METHOD FB_init : BOOL
VAR_INPUT
	bInitRetains : BOOL; // if TRUE, the retain variables are initialized (warm start / cold start)
	bInCopyCode : BOOL;  // if TRUE, the instance afterwards gets moved into the copy code (online change)
END_VAR
AddInput('ipRefContour', ipRefContour);
AddInput('ipContours', ipContours);
AddParameter('fDissimilarityThreshold', fDissimilarityThreshold);
AddParameter('eComparisonMethod', eComparisonMethod);
AddParameter('fAreaFactor', fAreaFactor);
AddParameter('fAbsPositionFactor', fAbsPositionFactor);
AddInput('hrPrev', hrPrev);
AddOutput('ipMatchIndexes', ipMatchIndexes);
AddOutput('ipDissimilarities', ipDissimilarities);
AddOutput('hresult', hresult);
END_METHOD

METHOD PUBLIC  Clone : I_Node
VAR
	pNode : POINTER TO Node_F_VN_MatchContours1vsNExp;
END_VAR
pNode := __NEW(Node_F_VN_MatchContours1vsNExp);
Clone := pNode^;
END_METHOD

METHOD PROTECTED OnExecute
hresult.Value := F_VN_MatchContours1vsNExp(
	ipRefContour := ipRefContour.Value,
    ipContours := ipContours.Value,
    ipMatchIndexes := ipMatchIndexes.Value,
    ipDissimilarities := ipDissimilarities.Value,
    fDissimilarityThreshold := fDissimilarityThreshold.Value,
    eComparisonMethod := eComparisonMethod.Value,
    fAreaFactor := fAreaFactor.Value,
    fAbsPositionFactor := fAbsPositionFactor.Value,
	hrPrev:= hrPrev.Value);
END_METHOD

METHOD PUBLIC PreExecutionCheck
VAR_INPUT
	Check : I_PreExecutionChecks;
END_VAR
Check.IsTrue(ipRefContour.IsValid, 'ipRefContour must be a valid container');
Check.IsTrue((ipRefContour.IsType(TC_GLOBAL_CONST_LIST.ContainerType_Vector_TcVnPoint2_DINT) OR
              ipRefContour.IsType(TC_GLOBAL_CONST_LIST.ContainerType_Vector_TcVnPoint2_REAL)),
              'ipRefContour contains incorrect type');
              
Check.IsTrue(ipContours.IsValid, 'ipContours must be a valid container');
Check.IsTrue(ipContours.IsType(TC_GLOBAL_CONST_LIST.ContainerType_Vector_Vector_TcVnPoint2_DINT), 'ipContours contains incorrect type');

Check.IsTrue(fAreaFactor.Value >= 0, 'fAreaFactor must be greater than or equal to 0');
Check.IsTrue(fAbsPositionFactor.Value >= 0, 'fAbsPositionFactor must be greater than or equal to 0');
END_METHOD

END_FUNCTION_BLOCK

// Nodes/Contour Analysis/Node_F_VN_MatchContoursExp
{attribute 'linkalways'}
{attribute 'no_explicit_call' := 'This FB is a CLASS and must be accessed using methods or properties'}
{attribute 'enable_dynamic_creation'}
FUNCTION_BLOCK Node_F_VN_MatchContoursExp EXTENDS VisionNode
VAR
    ipContour1 : _ITcVnContainer;
    ipContour2 : _ITcVnContainer;
    eComparisonMethod : _ETcVnContoursMatchComparisonMethod(ETcVnContoursMatchComparisonMethod.TCVN_CMCM_CONTOURS_MATCH_I1);
    fDissimilarity : _LREAL(0.0);
    fAreaFactor : _LREAL(0);
    fAbsPositionFactor : _LREAL(0);
    fRelPositionFactor : _LREAL(0);
    fNumDiffFactor : _LREAL(0);
    hrPrev : _HRESULT(S_OK);
    hresult : _HRESULT(S_OK);
END_VAR

METHOD FB_init : BOOL
VAR_INPUT
    bInitRetains : BOOL;
    bInCopyCode : BOOL;
END_VAR
AddInput('ipContour1', ipContour1);
AddInput('ipContour2', ipContour2);
AddParameter('eComparisonMethod', eComparisonMethod);
AddOutput('fDissimilarity', fDissimilarity);
AddParameter('fAreaFactor', fAreaFactor);
AddParameter('fAbsPositionFactor', fAbsPositionFactor);
AddParameter('fRelPositionFactor', fRelPositionFactor);
AddParameter('fNumDiffFactor', fNumDiffFactor);
AddInput('hrPrev', hrPrev);
AddOutput('hresult', hresult);
END_METHOD

METHOD PUBLIC Clone : I_Node
VAR
    pNode : POINTER TO Node_F_VN_MatchContoursExp;
END_VAR
pNode := __NEW(Node_F_VN_MatchContoursExp);
Clone := pNode^;
END_METHOD

METHOD PROTECTED OnExecute
hresult.Value := F_VN_MatchContoursExp(
    ipContour1 := ipContour1.Value,
    ipContour2 := ipContour2.Value,
    eComparisonMethod := eComparisonMethod.Value,
    fDissimilarity := fDissimilarity.Value,
    fAreaFactor := fAreaFactor.Value,
    fAbsPositionFactor := fAbsPositionFactor.Value,
    fRelPositionFactor := fRelPositionFactor.Value,
    fNumDiffFactor := fNumDiffFactor.Value,
    hrPrev := hrPrev.Value);
END_METHOD

METHOD PUBLIC PreExecutionCheck
VAR_INPUT
    Check : I_PreExecutionChecks;
END_VAR
Check.IsTrue(ipContour1.IsValid, 'ipContour1 must contain a container');
Check.IsTrue(ipContour2.IsValid, 'ipContour2 must contain a container');
Check.IsTrue(ipContour1.IsType(TC_GLOBAL_CONST_LIST.ContainerType_Vector_TcVnPoint2_DINT) OR
             ipContour1.IsType(TC_GLOBAL_CONST_LIST.ContainerType_Vector_TcVnPoint2_REAL) OR
             ipContour1.IsType(TC_GLOBAL_CONST_LIST.ContainerType_Vector_Vector_TcVnPoint2_DINT), 'Unsupported contour container type');
Check.IsTrue(ContainersHaveMatchingTypes(ipContour1.Value, ipContour2.Value), 'Contours must have matching container types');
Check.IsTrue((eComparisonMethod.Value = ETcVnContoursMatchComparisonMethod.TCVN_CMCM_CONTOURS_MATCH_I1) OR
             (eComparisonMethod.Value = ETcVnContoursMatchComparisonMethod.TCVN_CMCM_CONTOURS_MATCH_I2) OR
             (eComparisonMethod.Value = ETcVnContoursMatchComparisonMethod.TCVN_CMCM_CONTOURS_MATCH_I3), 'Unsupported eComparisonMethod');
END_METHOD

END_FUNCTION_BLOCK

// Nodes/Contour Analysis/Node_F_VN_UprightBoundingRectangle
{attribute 'linkalways'} 
{attribute 'no_explicit_call' := 'This FB is a CLASS and must be accessed using methods or properties'}
{attribute 'enable_dynamic_creation'}
FUNCTION_BLOCK Node_F_VN_UprightBoundingRectangle EXTENDS VisionNode
VAR
    ipPointSet : _ITcVnContainer;
    stRectangle : _TcVnRectangle_UDINT;
    hrPrev : _HRESULT(S_OK);
	hresult : _HRESULT(S_OK);
END_VAR

METHOD FB_init : BOOL
VAR_INPUT
	bInitRetains : BOOL; // if TRUE, the retain variables are initialized (warm start / cold start)
	bInCopyCode : BOOL;  // if TRUE, the instance afterwards gets moved into the copy code (online change)
END_VAR
AddInput('ipPointSet', ipPointSet);
AddInput('hrPrev', hrPrev);
AddOutput('stRectangle', stRectangle);
AddOutput('hresult',hresult);
END_METHOD

METHOD PUBLIC  Clone : I_Node
VAR
	pNode : POINTER TO Node_F_VN_UprightBoundingRectangle;
END_VAR
pNode := __NEW(Node_F_VN_UprightBoundingRectangle);
Clone := pNode^;
END_METHOD

METHOD PROTECTED OnExecute
hresult.Value := F_VN_UprightBoundingRectangle(
	ipPointSet := ipPointSet.Value,
    stRectangle := stRectangle.Value,
	hrPrev:= hrPrev.Value);
END_METHOD

METHOD PUBLIC PreExecutionCheck
VAR_INPUT
	Check : I_PreExecutionChecks;
END_VAR
Check.IsTrue(ipPointSet.IsValid, 'ipPointSet must be a valid container');
Check.IsTrue((ipPointSet.IsType(TC_GLOBAL_CONST_LIST.ContainerType_Vector_TcVnPoint2_DINT) OR
              ipPointSet.IsType(TC_GLOBAL_CONST_LIST.ContainerType_Vector_TcVnPoint2_REAL)),
              'ipPointSet contains incorrect type');
END_METHOD

END_FUNCTION_BLOCK

// Nodes/Drawing/Node_F_VN_DrawArrow
{attribute 'linkalways'} 
{attribute 'no_explicit_call' := 'This FB is a CLASS and must be accessed using methods or properties'}
{attribute 'enable_dynamic_creation'}
FUNCTION_BLOCK Node_F_VN_DrawArrow EXTENDS VisionNode
VAR
    nX1 : _UDINT(0);
    nY1 : _UDINT(0);
    nX2 : _UDINT(0);
    nY2 : _UDINT(0);
    ipDestImage : _ITcVnImage;
    aColor : _TcVnVector4_LREAL;
    nThickness : _DINT(1);
    bDoubleHead : _BOOL(FALSE);
    hrPrev : _HRESULT(S_OK);
	hresult : _HRESULT(S_OK);
END_VAR

METHOD FB_init : BOOL
VAR_INPUT
	bInitRetains : BOOL; // if TRUE, the retain variables are initialized (warm start / cold start)
	bInCopyCode : BOOL;  // if TRUE, the instance afterwards gets moved into the copy code (online change)
END_VAR
AddParameter('nX1', nX1);
AddParameter('nY1', nY1);
AddParameter('nX2', nX2);
AddParameter('nY2', nY2);
AddInput('ipDestImage', ipDestImage);
AddInput('aColor', aColor);
AddParameter('nThickness', nThickness);
AddParameter('bDoubleHead', bDoubleHead);
AddInput('hrPrev', hrPrev);
AddOutput('ipDestImage', ipDestImage);
AddOutput('hresult',hresult);
END_METHOD

METHOD PUBLIC  Clone : I_Node
VAR
	pNode : POINTER TO Node_F_VN_DrawArrow;
END_VAR
pNode := __NEW(Node_F_VN_DrawArrow);
Clone := pNode^;
END_METHOD

METHOD PROTECTED OnExecute
hresult.Value := F_VN_DrawArrow(
    nX1 := nX1.Value,
    nY1 := nY1.Value,
    nX2 := nX2.Value,
    nY2 := nY2.Value,
	ipDestImage := ipDestImage.Value,
    aColor := aColor.Value,
    nThickness := nThickness.Value,
    bDoubleHead := bDoubleHead.Value,
	hrPrev:= hrPrev.Value);
END_METHOD

METHOD PUBLIC PreExecutionCheck
VAR_INPUT
	Check : I_PreExecutionChecks;
END_VAR
Check.IsTrue(ipDestImage.IsValid, 'ipDestImage must contain an image');
Check.IsTrue(nThickness.Value >= 1, 'nThickness must be greater than or equal to 1');
END_METHOD

END_FUNCTION_BLOCK

// Nodes/Drawing/Node_F_VN_DrawArrow_TcVnVector4_DINT
{attribute 'linkalways'} 
{attribute 'no_explicit_call' := 'This FB is a CLASS and must be accessed using methods or properties'}
{attribute 'enable_dynamic_creation'}
FUNCTION_BLOCK Node_F_VN_DrawArrow_TcVnVector4_DINT EXTENDS VisionNode
VAR
    aLine : _TcVnVector4_DINT;
    ipDestImage : _ITcVnImage;
    aColor : _TcVnVector4_LREAL;
    nThickness : _DINT(1);
    bDoubleHead : _BOOL(FALSE);
    hrPrev : _HRESULT(S_OK);
	hresult : _HRESULT(S_OK);
END_VAR

METHOD FB_init : BOOL
VAR_INPUT
	bInitRetains : BOOL; // if TRUE, the retain variables are initialized (warm start / cold start)
	bInCopyCode : BOOL;  // if TRUE, the instance afterwards gets moved into the copy code (online change)
END_VAR
AddInput('aLine', aLine);
AddInput('ipDestImage', ipDestImage);
AddInput('aColor', aColor);
AddParameter('nThickness', nThickness);
AddParameter('bDoubleHead', bDoubleHead);
AddInput('hrPrev', hrPrev);
AddOutput('ipDestImage', ipDestImage);
AddOutput('hresult',hresult);
END_METHOD

METHOD PUBLIC  Clone : I_Node
VAR
	pNode : POINTER TO Node_F_VN_DrawArrow_TcVnVector4_DINT;
END_VAR
pNode := __NEW(Node_F_VN_DrawArrow_TcVnVector4_DINT);
Clone := pNode^;
END_METHOD

METHOD PROTECTED OnExecute
hresult.Value := F_VN_DrawArrow_TcVnVector4_DINT(
    aLine := aLine.Value,
	ipDestImage := ipDestImage.Value,
    aColor := aColor.Value,
    nThickness := nThickness.Value,
    bDoubleHead := bDoubleHead.Value,
	hrPrev:= hrPrev.Value);
END_METHOD

METHOD PUBLIC PreExecutionCheck
VAR_INPUT
	Check : I_PreExecutionChecks;
END_VAR
Check.IsTrue(ipDestImage.IsValid, 'ipDestImage must contain an image');
Check.IsTrue(nThickness.Value >= 1, 'nThickness must be greater than or equal to 1');
END_METHOD

END_FUNCTION_BLOCK

// Nodes/Drawing/Node_F_VN_DrawArrowExp
{attribute 'linkalways'} 
{attribute 'no_explicit_call' := 'This FB is a CLASS and must be accessed using methods or properties'}
{attribute 'enable_dynamic_creation'}
FUNCTION_BLOCK Node_F_VN_DrawArrowExp EXTENDS VisionNode
VAR
    nX1 : _UDINT(0);
    nY1 : _UDINT(0);
    nX2 : _UDINT(0);
    nY2 : _UDINT(0);
    ipDestImage : _ITcVnImage;
    aColor : _TcVnVector4_LREAL;
    nThickness : _DINT(1);
    bDoubleHead : _BOOL(FALSE);
    eLineType : _ETcVnLineType(ETcVnLineType.TCVN_LT_4_CONNECTED);
    nShift : _UDINT(0);
    fTipLength : _LREAL(0.0);
    hrPrev : _HRESULT(S_OK);
	hresult : _HRESULT(S_OK);
END_VAR

METHOD FB_init : BOOL
VAR_INPUT
	bInitRetains : BOOL; // if TRUE, the retain variables are initialized (warm start / cold start)
	bInCopyCode : BOOL;  // if TRUE, the instance afterwards gets moved into the copy code (online change)
END_VAR
AddParameter('nX1', nX1);
AddParameter('nY1', nY1);
AddParameter('nX2', nX2);
AddParameter('nY2', nY2);
AddInput('ipDestImage', ipDestImage);
AddInput('aColor', aColor);
AddParameter('nThickness', nThickness);
AddParameter('bDoubleHead', bDoubleHead);
AddParameter('eLineType', eLineType);
AddParameter('nShift', nShift);
AddParameter('fTipLength', fTipLength);
AddInput('hrPrev', hrPrev);
AddOutput('ipDestImage', ipDestImage);
AddOutput('hresult', hresult);
END_METHOD

METHOD PUBLIC  Clone : I_Node
VAR
	pNode : POINTER TO Node_F_VN_DrawArrowExp;
END_VAR
pNode := __NEW(Node_F_VN_DrawArrowExp);
Clone := pNode^;
END_METHOD

METHOD PROTECTED OnExecute
hresult.Value := F_VN_DrawArrowExp(
    nX1 := nX1.Value,
    nY1 := nY1.Value,
    nX2 := nX2.Value,
    nY2 := nY2.Value,
	ipDestImage := ipDestImage.Value,
    aColor := aColor.Value,
    nThickness := nThickness.Value,
    bDoubleHead := bDoubleHead.Value,
    eLineType := eLineType.Value,
    nShift := nShift.Value,
    fTipLength := fTipLength.Value,
	hrPrev:= hrPrev.Value);
END_METHOD

METHOD PUBLIC PreExecutionCheck
VAR_INPUT
	Check : I_PreExecutionChecks;
END_VAR
Check.IsTrue(ipDestImage.IsValid, 'ipDestImage must contain an image');
Check.IsTrue(nThickness.Value >= 1, 'nThickness must be greater than or equal to 1');
END_METHOD

END_FUNCTION_BLOCK

// Nodes/Drawing/Node_F_VN_DrawArrowExp_TcVnVector4_DINT
{attribute 'linkalways'} 
{attribute 'no_explicit_call' := 'This FB is a CLASS and must be accessed using methods or properties'}
{attribute 'enable_dynamic_creation'}
FUNCTION_BLOCK Node_F_VN_DrawArrowExp_TcVnVector4_DINT EXTENDS VisionNode
VAR
    aLine : _TcVnVector4_DINT;
    ipDestImage : _ITcVnImage;
    aColor : _TcVnVector4_LREAL;
    nThickness : _DINT(1);
    bDoubleHead : _BOOL(FALSE);
    eLineType : _ETcVnLineType(ETcVnLineType.TCVN_LT_4_CONNECTED);
    nShift : _UDINT(0);
    fTipLength : _LREAL(0.0);
    hrPrev : _HRESULT(S_OK);
	hresult : _HRESULT(S_OK);
END_VAR

METHOD FB_init : BOOL
VAR_INPUT
	bInitRetains : BOOL; // if TRUE, the retain variables are initialized (warm start / cold start)
	bInCopyCode : BOOL;  // if TRUE, the instance afterwards gets moved into the copy code (online change)
END_VAR
AddInput('aLine', aLine);
AddInput('ipDestImage', ipDestImage);
AddInput('aColor', aColor);
AddParameter('nThickness', nThickness);
AddParameter('bDoubleHead', bDoubleHead);
AddParameter('eLineType', eLineType);
AddParameter('nShift', nShift);
AddParameter('fTipLength', fTipLength);
AddInput('hrPrev', hrPrev);
AddOutput('ipDestImage', ipDestImage);
AddOutput('hresult', hresult);
END_METHOD

METHOD PUBLIC  Clone : I_Node
VAR
	pNode : POINTER TO Node_F_VN_DrawArrowExp_TcVnVector4_DINT;
END_VAR
pNode := __NEW(Node_F_VN_DrawArrowExp_TcVnVector4_DINT);
Clone := pNode^;
END_METHOD

METHOD PROTECTED OnExecute
hresult.Value := F_VN_DrawArrowExp_TcVnVector4_DINT(
    aLine := aLine.Value,
	ipDestImage := ipDestImage.Value,
    aColor := aColor.Value,
    nThickness := nThickness.Value,
    bDoubleHead := bDoubleHead.Value,
    eLineType := eLineType.Value,
    nShift := nShift.Value,
    fTipLength := fTipLength.Value,
	hrPrev:= hrPrev.Value);
END_METHOD

METHOD PUBLIC PreExecutionCheck
VAR_INPUT
	Check : I_PreExecutionChecks;
END_VAR
Check.IsTrue(ipDestImage.IsValid, 'ipDestImage must contain an image');
Check.IsTrue(nThickness.Value >= 1, 'nThickness must be greater than or equal to 1');
END_METHOD

END_FUNCTION_BLOCK

// Nodes/Drawing/Node_F_VN_DrawCircle
{attribute 'linkalways'} 
{attribute 'no_explicit_call' := 'This FB is a CLASS and must be accessed using methods or properties'}
{attribute 'enable_dynamic_creation'}
FUNCTION_BLOCK Node_F_VN_DrawCircle EXTENDS VisionNode
VAR
    nCenterX : _UDINT(0);
    nCenterY : _UDINT(0);
    nRadius : _UDINT(0);
    ipDestImage : _ITcVnImage;
    aColor : _TcVnVector4_LREAL;
    nThickness : _DINT(1);
    hrPrev : _HRESULT(S_OK);
	hresult : _HRESULT(S_OK);
END_VAR

METHOD FB_init : BOOL
VAR_INPUT
	bInitRetains : BOOL; // if TRUE, the retain variables are initialized (warm start / cold start)
	bInCopyCode : BOOL;  // if TRUE, the instance afterwards gets moved into the copy code (online change)
END_VAR
AddParameter('nCenterX', nCenterX);
AddParameter('nCenterY', nCenterY);
AddParameter('nRadius', nRadius);
AddInput('ipDestImage', ipDestImage);
AddInput('aColor', aColor);
AddParameter('nThickness', nThickness);
AddInput('hrPrev', hrPrev);
AddOutput('ipDestImage', ipDestImage);
AddOutput('hresult',hresult);
END_METHOD

METHOD PUBLIC  Clone : I_Node
VAR
	pNode : POINTER TO Node_F_VN_DrawCircle;
END_VAR
pNode := __NEW(Node_F_VN_DrawCircle);
Clone := pNode^;
END_METHOD

METHOD PROTECTED OnExecute
hresult.Value := F_VN_DrawCircle(
    nCenterX := nCenterX.Value,
    nCenterY := nCenterY.Value,
    nRadius := nRadius.Value,
	ipDestImage := ipDestImage.Value,
    aColor := aColor.Value,
    nThickness := nThickness.Value,
	hrPrev:= hrPrev.Value);
END_METHOD

METHOD PUBLIC PreExecutionCheck
VAR_INPUT
	Check : I_PreExecutionChecks;
END_VAR
Check.IsTrue(ipDestImage.IsValid, 'ipDestImage must contain an image');
Check.IsTrue(nThickness.Value <> 0, 'nThickness must be non-zero');
END_METHOD

END_FUNCTION_BLOCK

// Nodes/Drawing/Node_F_VN_DrawCircleExp
{attribute 'linkalways'} 
{attribute 'no_explicit_call' := 'This FB is a CLASS and must be accessed using methods or properties'}
{attribute 'enable_dynamic_creation'}
FUNCTION_BLOCK Node_F_VN_DrawCircleExp EXTENDS VisionNode
VAR
    nCenterX : _UDINT(0);
    nCenterY : _UDINT(0);
    nRadius : _UDINT(0);
    ipDestImage : _ITcVnImage;
    aColor : _TcVnVector4_LREAL;
    nThickness : _DINT(1);
    eLineType : _ETcVnLineType(ETcVnLineType.TCVN_LT_4_CONNECTED);
    hrPrev : _HRESULT(S_OK);
	hresult : _HRESULT(S_OK);
END_VAR

METHOD FB_init : BOOL
VAR_INPUT
	bInitRetains : BOOL; // if TRUE, the retain variables are initialized (warm start / cold start)
	bInCopyCode : BOOL;  // if TRUE, the instance afterwards gets moved into the copy code (online change)
END_VAR
AddParameter('nCenterX', nCenterX);
AddParameter('nCenterY', nCenterY);
AddParameter('nRadius', nRadius);
AddInput('ipDestImage', ipDestImage);
AddInput('aColor', aColor);
AddParameter('nThickness', nThickness);
AddParameter('eLineType', eLineType);
AddInput('hrPrev', hrPrev);
AddOutput('ipDestImage', ipDestImage);
AddOutput('hresult',hresult);
END_METHOD

METHOD PUBLIC  Clone : I_Node
VAR
	pNode : POINTER TO Node_F_VN_DrawCircleExp;
END_VAR
pNode := __NEW(Node_F_VN_DrawCircleExp);
Clone := pNode^;
END_METHOD

METHOD PROTECTED OnExecute
hresult.Value := F_VN_DrawCircleExp(
    nCenterX := nCenterX.Value,
    nCenterY := nCenterY.Value,
    nRadius := nRadius.Value,
	ipDestImage := ipDestImage.Value,
    aColor := aColor.Value,
    nThickness := nThickness.Value,
    eLineType := eLineType.Value,
	hrPrev:= hrPrev.Value);
END_METHOD

METHOD PUBLIC PreExecutionCheck
VAR_INPUT
	Check : I_PreExecutionChecks;
END_VAR
Check.IsTrue(ipDestImage.IsValid, 'ipDestImage must contain an image');
Check.IsTrue(nThickness.Value <> 0, 'nThickness must be non-zero');
END_METHOD

END_FUNCTION_BLOCK

// Nodes/Drawing/Node_F_VN_DrawCircles
{attribute 'linkalways'} 
{attribute 'no_explicit_call' := 'This FB is a CLASS and must be accessed using methods or properties'}
{attribute 'enable_dynamic_creation'}
FUNCTION_BLOCK Node_F_VN_DrawCircles EXTENDS VisionNode
VAR
    ipCircles : _ITcVnContainer;
    nCircleIndex : _DINT(0);
    ipDestImage : _ITcVnImage;
    aColor : _TcVnVector4_LREAL;
    nThickness : _DINT(1);
    hrPrev : _HRESULT(S_OK);
	hresult : _HRESULT(S_OK);
END_VAR

METHOD FB_init : BOOL
VAR_INPUT
	bInitRetains : BOOL; // if TRUE, the retain variables are initialized (warm start / cold start)
	bInCopyCode : BOOL;  // if TRUE, the instance afterwards gets moved into the copy code (online change)
END_VAR
AddInput('ipCircles', ipCircles);
AddParameter('nCircleIndex', nCircleIndex);
AddInput('ipDestImage', ipDestImage);
AddInput('aColor', aColor);
AddParameter('nThickness', nThickness);
AddInput('hrPrev', hrPrev);
AddOutput('ipDestImage', ipDestImage);
AddOutput('hresult',hresult);
END_METHOD

METHOD PUBLIC  Clone : I_Node
VAR
	pNode : POINTER TO Node_F_VN_DrawCircles
;
END_VAR
pNode := __NEW(Node_F_VN_DrawCircles);
Clone := pNode^;
END_METHOD

METHOD PROTECTED OnExecute
hresult.Value := F_VN_DrawCircles(
    ipCircles := ipCircles.Value,
    nCircleIndex := nCircleIndex.Value,
	ipDestImage := ipDestImage.Value,
    aColor := aColor.Value,
    nThickness := nThickness.Value,
	hrPrev:= hrPrev.Value);
END_METHOD

METHOD PUBLIC PreExecutionCheck
VAR_INPUT
	Check : I_PreExecutionChecks;
END_VAR
VAR
    containerElements : ULINT;
    maxIndexNumber : ULINT;
END_VAR
Check.IsTrue(ipCircles.IsValid, 'ipCircles must be a valid container');
Check.IsTrue(ipCircles.IsType(TC_GLOBAL_CONST_LIST.ContainerType_Vector_TcVnVector3_REAL), 'ipCircles contains incorrect type');

Check.IsTrue(ipCircles.TryGetElementNum(containerElements) AND (containerElements > 0), 'ipCircles is empty');

IF Check.Failed THEN
    RETURN;
END_IF

maxIndexNumber := containerElements - 1;

IF (nCircleIndex.Value > -1) THEN
    Check.IsTrue((DINT_TO_ULINT(nCircleIndex.Value) <= maxIndexNumber), 'nCircleIndex out of range.');
END_IF

Check.IsTrue(ipDestImage.IsValid, 'ipDestImage must contain an image');
Check.IsTrue(nThickness.Value <> 0, 'nThickness must be non-zero');
END_METHOD

END_FUNCTION_BLOCK

// Nodes/Drawing/Node_F_VN_DrawCirclesExp
{attribute 'linkalways'} 
{attribute 'no_explicit_call' := 'This FB is a CLASS and must be accessed using methods or properties'}
{attribute 'enable_dynamic_creation'}
FUNCTION_BLOCK Node_F_VN_DrawCirclesExp EXTENDS VisionNode
VAR
    ipCircles : _ITcVnContainer;
    nCircleIndex : _DINT(0);
    ipDestImage : _ITcVnImage;
    aColor : _TcVnVector4_LREAL;
    nThickness : _DINT(1);
    eLineType : _ETcVnLineType(ETcVnLineType.TCVN_LT_4_CONNECTED);
    hrPrev : _HRESULT(S_OK);
	hresult : _HRESULT(S_OK);
END_VAR

METHOD FB_init : BOOL
VAR_INPUT
	bInitRetains : BOOL; // if TRUE, the retain variables are initialized (warm start / cold start)
	bInCopyCode : BOOL;  // if TRUE, the instance afterwards gets moved into the copy code (online change)
END_VAR
AddInput('ipCircles', ipCircles);
AddParameter('nCircleIndex', nCircleIndex);
AddInput('ipDestImage', ipDestImage);
AddInput('aColor', aColor);
AddParameter('nThickness', nThickness);
AddParameter('eLineType', eLineType);
AddInput('hrPrev', hrPrev);
AddOutput('ipDestImage', ipDestImage);
AddOutput('hresult',hresult);
END_METHOD

METHOD PUBLIC  Clone : I_Node
VAR
	pNode : POINTER TO Node_F_VN_DrawCirclesExp
;
END_VAR
pNode := __NEW(Node_F_VN_DrawCirclesExp);
Clone := pNode^;
END_METHOD

METHOD PROTECTED OnExecute
hresult.Value := F_VN_DrawCirclesExp(
    ipCircles := ipCircles.Value,
    nCircleIndex := nCircleIndex.Value,
	ipDestImage := ipDestImage.Value,
    aColor := aColor.Value,
    nThickness := nThickness.Value,
    eLineType := eLineType.Value,
	hrPrev:= hrPrev.Value);
END_METHOD

METHOD PUBLIC PreExecutionCheck
VAR_INPUT
	Check : I_PreExecutionChecks;
END_VAR
VAR
    containerElements : ULINT;
    maxIndexNumber : ULINT;
END_VAR
Check.IsTrue(ipCircles.IsValid, 'ipCircles must be a valid container');
Check.IsTrue(ipCircles.IsType(TC_GLOBAL_CONST_LIST.ContainerType_Vector_TcVnVector3_REAL), 'ipCircles contains incorrect type');

Check.IsTrue(ipCircles.TryGetElementNum(containerElements) AND (containerElements > 0), 'ipCircles is empty');

IF Check.Failed THEN
    RETURN;
END_IF

maxIndexNumber := containerElements - 1;

IF (nCircleIndex.Value > -1) THEN
    Check.IsTrue((DINT_TO_ULINT(nCircleIndex.Value) <= maxIndexNumber), 'nCircleIndex out of range.');
END_IF

Check.IsTrue(ipDestImage.IsValid, 'ipDestImage must contain an image');
Check.IsTrue(nThickness.Value <> 0, 'nThickness must be non-zero');
END_METHOD

END_FUNCTION_BLOCK

// Nodes/Drawing/Node_F_VN_DrawCircularArc
{attribute 'linkalways'} 
{attribute 'no_explicit_call' := 'This FB is a CLASS and must be accessed using methods or properties'}
{attribute 'enable_dynamic_creation'}
FUNCTION_BLOCK Node_F_VN_DrawCircularArc EXTENDS VisionNode
VAR
    stCircularArc : _TcVnCircularArc;
    ipDestImage : _ITcVnImage;
    aColor : _TcVnVector4_LREAL;
    nThickness : _DINT(1);
    hrPrev : _HRESULT(S_OK);
	hresult : _HRESULT(S_OK);
END_VAR

METHOD FB_init : BOOL
VAR_INPUT
	bInitRetains : BOOL; // if TRUE, the retain variables are initialized (warm start / cold start)
	bInCopyCode : BOOL;  // if TRUE, the instance afterwards gets moved into the copy code (online change)
END_VAR
AddInput('stCircularArc', stCircularArc);
AddInput('ipDestImage', ipDestImage);
AddInput('aColor', aColor);
AddParameter('nThickness', nThickness);
AddInput('hrPrev', hrPrev);
AddOutput('ipDestImage', ipDestImage);
AddOutput('hresult',hresult);
END_METHOD

METHOD PUBLIC  Clone : I_Node
VAR
	pNode : POINTER TO Node_F_VN_DrawCircularArc;
END_VAR
pNode := __NEW(Node_F_VN_DrawCircularArc);
Clone := pNode^;
END_METHOD

METHOD PROTECTED OnExecute
hresult.Value := F_VN_DrawCircularArc(
    stCircularArc := stCircularArc.Value,
	ipDestImage := ipDestImage.Value,
    aColor := aColor.Value,
    nThickness := nThickness.Value,
	hrPrev:= hrPrev.Value);
END_METHOD

METHOD PUBLIC PreExecutionCheck
VAR_INPUT
	Check : I_PreExecutionChecks;
END_VAR
Check.IsTrue(ipDestImage.IsValid, 'ipDestImage must contain an image');
Check.IsTrue(nThickness.Value <> 0, 'nThickness must be non-zero');
END_METHOD

END_FUNCTION_BLOCK

// Nodes/Drawing/Node_F_VN_DrawCircularArcExp
{attribute 'linkalways'} 
{attribute 'no_explicit_call' := 'This FB is a CLASS and must be accessed using methods or properties'}
{attribute 'enable_dynamic_creation'}
FUNCTION_BLOCK Node_F_VN_DrawCircularArcExp EXTENDS VisionNode
VAR
    stCircularArc : _TcVnCircularArc;
    ipDestImage : _ITcVnImage;
    aColor : _TcVnVector4_LREAL;
    nThickness : _DINT(1);
    eLineType : _ETcVnLineType(ETcVnLineType.TCVN_LT_4_CONNECTED);
    hrPrev : _HRESULT(S_OK);
	hresult : _HRESULT(S_OK);
END_VAR

METHOD FB_init : BOOL
VAR_INPUT
	bInitRetains : BOOL; // if TRUE, the retain variables are initialized (warm start / cold start)
	bInCopyCode : BOOL;  // if TRUE, the instance afterwards gets moved into the copy code (online change)
END_VAR
AddInput('stCircularArc', stCircularArc);
AddInput('ipDestImage', ipDestImage);
AddInput('aColor', aColor);
AddParameter('nThickness', nThickness);
AddParameter('eLineType', eLineType);
AddInput('hrPrev', hrPrev);
AddOutput('ipDestImage', ipDestImage);
AddOutput('hresult',hresult);
END_METHOD

METHOD PUBLIC  Clone : I_Node
VAR
	pNode : POINTER TO Node_F_VN_DrawCircularArcExp;
END_VAR
pNode := __NEW(Node_F_VN_DrawCircularArcExp);
Clone := pNode^;
END_METHOD

METHOD PROTECTED OnExecute
hresult.Value := F_VN_DrawCircularArcExp(
    stCircularArc := stCircularArc.Value,
	ipDestImage := ipDestImage.Value,
    aColor := aColor.Value,
    nThickness := nThickness.Value,
    eLineType := eLineType.Value,
	hrPrev:= hrPrev.Value);
END_METHOD

METHOD PUBLIC PreExecutionCheck
VAR_INPUT
	Check : I_PreExecutionChecks;
END_VAR
Check.IsTrue(ipDestImage.IsValid, 'ipDestImage must contain an image');
Check.IsTrue(nThickness.Value <> 0, 'nThickness must be non-zero');
END_METHOD

END_FUNCTION_BLOCK

// Nodes/Drawing/Node_F_VN_DrawComponents
{attribute 'linkalways'} 
{attribute 'no_explicit_call' := 'This FB is a CLASS and must be accessed using methods or properties'}
{attribute 'enable_dynamic_creation'}
FUNCTION_BLOCK Node_F_VN_DrawComponents EXTENDS VisionNode
VAR
    ipLabelImage : _ITcVnImage;
    nLabelID : _DINT(0);
    ipDestImage : _ITcVnImage;
    bShowLabelID : _BOOL(FALSE);
    hrPrev : _HRESULT(S_OK);
	hresult : _HRESULT(S_OK);
END_VAR

METHOD FB_init : BOOL
VAR_INPUT
	bInitRetains : BOOL; // if TRUE, the retain variables are initialized (warm start / cold start)
	bInCopyCode : BOOL;  // if TRUE, the instance afterwards gets moved into the copy code (online change)
END_VAR
AddInput('ipLabelImage', ipLabelImage);
AddParameter('nLabelID', nLabelID);
AddParameter('bShowLabelID', bShowLabelID);
AddInput('hrPrev', hrPrev);
AddOutput('ipDestImage', ipDestImage);
AddOutput('hresult',hresult);
END_METHOD

METHOD PUBLIC  Clone : I_Node
VAR
	pNode : POINTER TO Node_F_VN_DrawComponents;
END_VAR
pNode := __NEW(Node_F_VN_DrawComponents);
Clone := pNode^;
END_METHOD

METHOD PROTECTED OnExecute
hresult.Value := F_VN_DrawComponents(
	ipLabelImage := ipLabelImage.Value,
    nLabelID := nLabelID.Value,
    ipDestImage := ipDestImage.Value,
    bShowLabelID := bShowLabelID.Value,
	hrPrev:= hrPrev.Value);
END_METHOD

METHOD PUBLIC PreExecutionCheck
VAR_INPUT
	Check : I_PreExecutionChecks;
END_VAR
Check.IsTrue(ipLabelImage.IsValid, 'ipLabelImage must contain an image');
Check.IsTrue(ipLabelImage.HasChannelCount(1), 'ipLabelImage must have 1 channel');
Check.IsTrue((ipLabelImage.IsPixelDepth(16)  OR
              ipLabelImage.IsPixelDepth(32)), 'ipLabelImage must have 16 or 32 bit pixel depth');
END_METHOD

END_FUNCTION_BLOCK

// Nodes/Drawing/Node_F_VN_DrawComponentsExp
{attribute 'linkalways'} 
{attribute 'no_explicit_call' := 'This FB is a CLASS and must be accessed using methods or properties'}
{attribute 'enable_dynamic_creation'}
FUNCTION_BLOCK Node_F_VN_DrawComponentsExp EXTENDS VisionNode
VAR
    ipLabelImage : _ITcVnImage;
    nLabelID : _DINT(0);
    ipDestImage : _ITcVnImage;
    bShowLabelID : _BOOL(FALSE);
    aColor : _TcVnVector4_LREAL;
    nThickness : _DINT(1);
    fFontScale : _LREAL(1.0);
    hrPrev : _HRESULT(S_OK);
	hresult : _HRESULT(S_OK);
END_VAR

METHOD FB_init : BOOL
VAR_INPUT
	bInitRetains : BOOL; // if TRUE, the retain variables are initialized (warm start / cold start)
	bInCopyCode : BOOL;  // if TRUE, the instance afterwards gets moved into the copy code (online change)
END_VAR
AddInput('ipLabelImage', ipLabelImage);
AddParameter('nLabelID', nLabelID);
AddInput('bShowLabelID', bShowLabelID);
AddInput('aColor', aColor);
AddParameter('nThickness', nThickness);
AddParameter('fFontScale', fFontScale);
AddInput('hrPrev', hrPrev);
AddOutput('ipDestImage', ipDestImage);
AddOutput('hresult',hresult);
END_METHOD

METHOD PUBLIC  Clone : I_Node
VAR
	pNode : POINTER TO Node_F_VN_DrawComponentsExp;
END_VAR
pNode := __NEW(Node_F_VN_DrawComponentsExp);
Clone := pNode^;
END_METHOD

METHOD PROTECTED OnExecute
hresult.Value := F_VN_DrawComponentsExp(
	ipLabelImage := ipLabelImage.Value,
    nLabelID := nLabelID.Value,
    ipDestImage := ipDestImage.Value,
    bShowLabelID := bShowLabelID.Value,
    aColor := aColor.Value,
    nThickness := nThickness.Value,
    fFontScale := fFontScale.Value,
	hrPrev:= hrPrev.Value);
END_METHOD

METHOD PUBLIC PreExecutionCheck
VAR_INPUT
	Check : I_PreExecutionChecks;
END_VAR
Check.IsTrue(ipLabelImage.IsValid, 'ipLabelImage must contain an image');
Check.IsTrue(ipLabelImage.HasChannelCount(1), 'ipLabelImage must have 1 channel');
Check.IsTrue((ipLabelImage.IsPixelDepth(16)  OR
              ipLabelImage.IsPixelDepth(32)), 'ipLabelImage must have 16 or 32 bit pixel depth');
Check.IsTrue(nThickness.Value >= 1, 'nThickness must be greater than or equal to 1');
END_METHOD

END_FUNCTION_BLOCK

// Nodes/Drawing/Node_F_VN_DrawContours
{attribute 'linkalways'} 
{attribute 'no_explicit_call' := 'This FB is a CLASS and must be accessed using methods or properties'}
{attribute 'enable_dynamic_creation'}
FUNCTION_BLOCK Node_F_VN_DrawContours EXTENDS VisionNode
VAR
    ipContours : _ITcVnContainer;
    nContourIndex : _DINT(0);
    ipDestImage : _ITcVnImage;
    aColor : _TcVnVector4_LREAL;
    nThickness : _DINT(1);
    hrPrev : _HRESULT(S_OK);
	hresult : _HRESULT(S_OK);
END_VAR

METHOD FB_init : BOOL
VAR_INPUT
	bInitRetains : BOOL; // if TRUE, the retain variables are initialized (warm start / cold start)
	bInCopyCode : BOOL;  // if TRUE, the instance afterwards gets moved into the copy code (online change)
END_VAR
AddInput('ipContours', ipContours);
AddParameter('nContourIndex', nContourIndex);
AddInput('ipDestImage', ipDestImage);
AddInput('aColor', aColor);
AddParameter('nThickness', nThickness);
AddInput('hrPrev', hrPrev);
AddOutput('ipDestImage', ipDestImage);
AddOutput('hresult',hresult);
END_METHOD

METHOD PUBLIC  Clone : I_Node
VAR
	pNode : POINTER TO Node_F_VN_DrawContours
;
END_VAR
pNode := __NEW(Node_F_VN_DrawContours);
Clone := pNode^;
END_METHOD

METHOD PROTECTED OnExecute
hresult.Value := F_VN_DrawContours(
    ipContours := ipContours.Value,
    nContourIndex := nContourIndex.Value,
	ipDestImage := ipDestImage.Value,
    aColor := aColor.Value,
    nThickness := nThickness.Value,
	hrPrev:= hrPrev.Value);
END_METHOD

METHOD PUBLIC PreExecutionCheck
VAR_INPUT
	Check : I_PreExecutionChecks;
END_VAR
VAR
    containerElements : ULINT;
    maxIndexNumber : ULINT;
END_VAR
Check.IsTrue(ipContours.IsValid, 'ipContours must be a valid container');
Check.IsTrue((ipContours.IsType(TC_GLOBAL_CONST_LIST.ContainerType_Vector_TcVnPoint2_DINT) OR
              ipContours.IsType(TC_GLOBAL_CONST_LIST.ContainerType_Vector_Vector_TcVnPoint2_DINT)),
              'ipContours contains incorrect type');

Check.IsTrue(ipDestImage.IsValid, 'ipDestImage must contain an image');
Check.IsTrue(nThickness.Value <> 0, 'nThickness must be non-zero');
END_METHOD

END_FUNCTION_BLOCK

// Nodes/Drawing/Node_F_VN_DrawContoursExp
{attribute 'linkalways'} 
{attribute 'no_explicit_call' := 'This FB is a CLASS and must be accessed using methods or properties'}
{attribute 'enable_dynamic_creation'}
FUNCTION_BLOCK Node_F_VN_DrawContoursExp EXTENDS VisionNode
VAR
    ipContours : _ITcVnContainer;
    nContourIndex : _DINT(0);
    ipDestImage : _ITcVnImage;
    aColor : _TcVnVector4_LREAL;
    nThickness : _DINT(1);
    eLineType : _ETcVnLineType(ETcVnLineType.TCVN_LT_4_CONNECTED);
    ipHierarchy : _ITcVnContainer;
    nMaxLevel : _DINT(0);
    aOffset : _TcVnPoint;
    hrPrev : _HRESULT(S_OK);
	hresult : _HRESULT(S_OK);
END_VAR

METHOD FB_init : BOOL
VAR_INPUT
	bInitRetains : BOOL; // if TRUE, the retain variables are initialized (warm start / cold start)
	bInCopyCode : BOOL;  // if TRUE, the instance afterwards gets moved into the copy code (online change)
END_VAR
AddInput('ipContours', ipContours);
AddParameter('nContourIndex', nContourIndex);
AddInput('ipDestImage', ipDestImage);
AddInput('aColor', aColor);
AddParameter('nThickness', nThickness);
AddParameter('eLineType', eLineType);
AddInput('ipHierarchy', ipHierarchy);
AddParameter('nMaxLevel', nMaxLevel);
AddInput('aOffset', aOffset);
AddInput('hrPrev', hrPrev);
AddOutput('ipDestImage', ipDestImage);
AddOutput('hresult',hresult);
END_METHOD

METHOD PUBLIC  Clone : I_Node
VAR
	pNode : POINTER TO Node_F_VN_DrawContoursExp
;
END_VAR
pNode := __NEW(Node_F_VN_DrawContoursExp);
Clone := pNode^;
END_METHOD

METHOD PROTECTED OnExecute
hresult.Value := F_VN_DrawContoursExp(
    ipContours := ipContours.Value,
    nContourIndex := nContourIndex.Value,
	ipDestImage := ipDestImage.Value,
    aColor := aColor.Value,
    nThickness := nThickness.Value,
    eLineType := eLineType.Value,
    ipHierarchy := ipHierarchy.Value,
    nMaxLevel := nMaxLevel.Value,
    aOffset := aOffset.Value,
	hrPrev:= hrPrev.Value);
END_METHOD

METHOD PUBLIC PreExecutionCheck
VAR_INPUT
	Check : I_PreExecutionChecks;
END_VAR
VAR
    containerElements : ULINT;
    maxIndexNumber : ULINT;
END_VAR
Check.IsTrue(ipContours.IsValid, 'ipContours must be a valid container');
Check.IsTrue((ipContours.IsType(TC_GLOBAL_CONST_LIST.ContainerType_Vector_TcVnPoint2_DINT) OR
              ipContours.IsType(TC_GLOBAL_CONST_LIST.ContainerType_Vector_Vector_TcVnPoint2_DINT)),
              'ipContours contains incorrect type');

Check.IsTrue(ipDestImage.IsValid, 'ipDestImage must contain an image');
Check.IsTrue(nThickness.Value <> 0, 'nThickness must be non-zero');
END_METHOD

END_FUNCTION_BLOCK

// Nodes/Drawing/Node_F_VN_DrawEllipse
{attribute 'linkalways'} 
{attribute 'no_explicit_call' := 'This FB is a CLASS and must be accessed using methods or properties'}
{attribute 'enable_dynamic_creation'}
FUNCTION_BLOCK Node_F_VN_DrawEllipse EXTENDS VisionNode
VAR
    stEllipse : _TcVnRotatedRectangle;
    ipDestImage : _ITcVnImage;
    aColor : _TcVnVector4_LREAL;
    nThickness : _DINT(1);
    hrPrev : _HRESULT(S_OK);
	hresult : _HRESULT(S_OK);
END_VAR

METHOD FB_init : BOOL
VAR_INPUT
	bInitRetains : BOOL; // if TRUE, the retain variables are initialized (warm start / cold start)
	bInCopyCode : BOOL;  // if TRUE, the instance afterwards gets moved into the copy code (online change)
END_VAR
AddInput('stEllipse', stEllipse);
AddInput('ipDestImage', ipDestImage);
AddInput('aColor', aColor);
AddInput('hrPrev', hrPrev);
AddOutput('ipDestImage', ipDestImage);
AddOutput('hresult',hresult);
AddParameter('nThickness', nThickness);
END_METHOD

METHOD PUBLIC  Clone : I_Node
VAR
	pNode : POINTER TO Node_F_VN_DrawEllipse;
END_VAR
pNode := __NEW(Node_F_VN_DrawEllipse);
Clone := pNode^;
END_METHOD

METHOD PROTECTED OnExecute
hresult.Value := F_VN_DrawEllipse(
    stEllipse := stEllipse.Value,
	ipDestImage := ipDestImage.Value,
    aColor := aColor.Value,
    nThickness := nThickness.Value,
	hrPrev:= hrPrev.Value);
END_METHOD

METHOD PUBLIC PreExecutionCheck
VAR_INPUT
	Check : I_PreExecutionChecks;
END_VAR
Check.IsTrue(ipDestImage.IsValid, 'ipDestImage must contain an image');
Check.IsTrue(nThickness.Value <> 0, 'nThickness must be non-zero');
END_METHOD

END_FUNCTION_BLOCK

// Nodes/Drawing/Node_F_VN_DrawEllipseExp
{attribute 'linkalways'} 
{attribute 'no_explicit_call' := 'This FB is a CLASS and must be accessed using methods or properties'}
{attribute 'enable_dynamic_creation'}
FUNCTION_BLOCK Node_F_VN_DrawEllipseExp EXTENDS VisionNode
VAR
    stEllipse : _TcVnRotatedRectangle;
    ipDestImage : _ITcVnImage;
    aColor : _TcVnVector4_LREAL;
    nThickness : _DINT(1);
    eLineType : _ETcVnLineType(ETcVnLineType.TCVN_LT_4_CONNECTED);
    hrPrev : _HRESULT(S_OK);
	hresult : _HRESULT(S_OK);
END_VAR

METHOD FB_init : BOOL
VAR_INPUT
	bInitRetains : BOOL; // if TRUE, the retain variables are initialized (warm start / cold start)
	bInCopyCode : BOOL;  // if TRUE, the instance afterwards gets moved into the copy code (online change)
END_VAR
AddInput('stEllipse', stEllipse);
AddInput('ipDestImage', ipDestImage);
AddInput('aColor', aColor);
AddParameter('nThickness', nThickness);
AddParameter('eLineType', eLineType);
AddInput('hrPrev', hrPrev);
AddOutput('ipDestImage', ipDestImage);
AddOutput('hresult',hresult);
END_METHOD

METHOD PUBLIC  Clone : I_Node
VAR
	pNode : POINTER TO Node_F_VN_DrawEllipseExp;
END_VAR
pNode := __NEW(Node_F_VN_DrawEllipseExp);
Clone := pNode^;
END_METHOD

METHOD PROTECTED OnExecute
hresult.Value := F_VN_DrawEllipseExp(
    stEllipse := stEllipse.Value,
	ipDestImage := ipDestImage.Value,
    aColor := aColor.Value,
    nThickness := nThickness.Value,
    eLineType := eLineType.Value,
	hrPrev:= hrPrev.Value);
END_METHOD

METHOD PUBLIC PreExecutionCheck
VAR_INPUT
	Check : I_PreExecutionChecks;
END_VAR
Check.IsTrue(ipDestImage.IsValid, 'ipDestImage must contain an image');
Check.IsTrue(nThickness.Value <> 0, 'nThickness must be non-zero');
END_METHOD

END_FUNCTION_BLOCK

// Nodes/Drawing/Node_F_VN_DrawKeypoints
{attribute 'linkalways'} 
{attribute 'no_explicit_call' := 'This FB is a CLASS and must be accessed using methods or properties'}
{attribute 'enable_dynamic_creation'}
FUNCTION_BLOCK Node_F_VN_DrawKeypoints EXTENDS VisionNode
VAR
    ipSrcImage : _ITcVnImage;
    ipKeyPoints : _ITcVnContainer;
    ipDestImage : _ITcVnImage;
    hrPrev : _HRESULT(S_OK);
	hresult : _HRESULT(S_OK);
END_VAR

METHOD FB_init : BOOL
VAR_INPUT
	bInitRetains : BOOL; // if TRUE, the retain variables are initialized (warm start / cold start)
	bInCopyCode : BOOL;  // if TRUE, the instance afterwards gets moved into the copy code (online change)
END_VAR
AddInput('ipSrcImage', ipSrcImage);
AddInput('ipKeyPoints', ipKeyPoints);
AddInput('hrPrev', hrPrev);
AddOutput('ipDestImage', ipDestImage);
AddOutput('hresult',hresult);
END_METHOD

METHOD PUBLIC  Clone : I_Node
VAR
	pNode : POINTER TO Node_F_VN_DrawKeypoints
;
END_VAR
pNode := __NEW(Node_F_VN_DrawKeypoints);
Clone := pNode^;
END_METHOD

METHOD PROTECTED OnExecute
hresult.Value := F_VN_DrawKeypoints(
    ipSrcImage := ipSrcImage.Value,
    ipKeyPoints := ipKeyPoints.Value,
	ipDestImage := ipDestImage.Value,
	hrPrev:= hrPrev.Value);
END_METHOD

METHOD PUBLIC PreExecutionCheck
VAR_INPUT
	Check : I_PreExecutionChecks;
END_VAR
Check.IsTrue(ipSrcImage.IsValid, 'ipSrcImage must contain an image');
Check.IsTrue(ipKeyPoints.IsType(TC_GLOBAL_CONST_LIST.ContainerType_Vector_TcVnKeyPoint), 'ipKeyPoints contains incorrect type');
END_METHOD

END_FUNCTION_BLOCK

// Nodes/Drawing/Node_F_VN_DrawKeypointsExp
{attribute 'linkalways'} 
{attribute 'no_explicit_call' := 'This FB is a CLASS and must be accessed using methods or properties'}
{attribute 'enable_dynamic_creation'}
FUNCTION_BLOCK Node_F_VN_DrawKeypointsExp EXTENDS VisionNode
VAR
    ipSrcImage : _ITcVnImage;
    ipKeyPoints : _ITcVnContainer;
    ipDestImage : _ITcVnImage;
    aColor : _TcVnVector4_LREAL;
    eFlags : _ETcVnDrawMatchesFlags(ETcVnDrawMatchesFlags.TCVN_DMF_DEFAULT);
    hrPrev : _HRESULT(S_OK);
	hresult : _HRESULT(S_OK);
END_VAR

METHOD FB_init : BOOL
VAR_INPUT
	bInitRetains : BOOL; // if TRUE, the retain variables are initialized (warm start / cold start)
	bInCopyCode : BOOL;  // if TRUE, the instance afterwards gets moved into the copy code (online change)
END_VAR
AddInput('ipSrcImage', ipSrcImage);
AddInput('ipKeyPoints', ipKeyPoints);
AddInput('aColor', aColor);
AddParameter('eFlags', eFlags);
AddInput('hrPrev', hrPrev);
AddOutput('ipDestImage', ipDestImage);
AddOutput('hresult',hresult);
END_METHOD

METHOD PUBLIC  Clone : I_Node
VAR
	pNode : POINTER TO Node_F_VN_DrawKeypointsExp
;
END_VAR
pNode := __NEW(Node_F_VN_DrawKeypointsExp);
Clone := pNode^;
END_METHOD

METHOD PROTECTED OnExecute
hresult.Value := F_VN_DrawKeypointsExp(
    ipSrcImage := ipSrcImage.Value,
    ipKeyPoints := ipKeyPoints.Value,
	ipDestImage := ipDestImage.Value,
    aColor := aColor.Value,
    eFlags := eFlags.Value,
	hrPrev:= hrPrev.Value);
END_METHOD

METHOD PUBLIC PreExecutionCheck
VAR_INPUT
	Check : I_PreExecutionChecks;
END_VAR
Check.IsTrue(ipSrcImage.IsValid, 'ipSrcImage must contain an image');
Check.IsTrue(ipSrcImage.IsPixelDepth(8), 'ipSrcImage must have 8 bit pixel depth');
Check.IsTrue(ipKeyPoints.IsType(TC_GLOBAL_CONST_LIST.ContainerType_Vector_TcVnKeyPoint), 'ipKeyPoints contains incorrect type');
END_METHOD

END_FUNCTION_BLOCK

// Nodes/Drawing/Node_F_VN_DrawLine
{attribute 'linkalways'} 
{attribute 'no_explicit_call' := 'This FB is a CLASS and must be accessed using methods or properties'}
{attribute 'enable_dynamic_creation'}
FUNCTION_BLOCK Node_F_VN_DrawLine EXTENDS VisionNode
VAR
    nX1 : _UDINT(0);
    nY1 : _UDINT(0);
    nX2 : _UDINT(0);
    nY2 : _UDINT(0);
    ipDestImage : _ITcVnImage;
    aColor : _TcVnVector4_LREAL;
    nThickness : _DINT(1);
    hrPrev : _HRESULT(S_OK);
	hresult : _HRESULT(S_OK);
END_VAR

METHOD FB_init : BOOL
VAR_INPUT
	bInitRetains : BOOL; // if TRUE, the retain variables are initialized (warm start / cold start)
	bInCopyCode : BOOL;  // if TRUE, the instance afterwards gets moved into the copy code (online change)
END_VAR
AddParameter('nX1', nX1);
AddParameter('nY1', nY1);
AddParameter('nX2', nX2);
AddParameter('nY2', nY2);
AddInput('ipDestImage', ipDestImage);
AddInput('aColor', aColor);
AddParameter('nThickness', nThickness);
AddInput('hrPrev', hrPrev);
AddOutput('ipDestImage', ipDestImage);
AddOutput('hresult',hresult);
END_METHOD

METHOD PUBLIC  Clone : I_Node
VAR
	pNode : POINTER TO Node_F_VN_DrawLine;
END_VAR
pNode := __NEW(Node_F_VN_DrawLine);
Clone := pNode^;
END_METHOD

METHOD PROTECTED OnExecute
hresult.Value := F_VN_DrawLine(
    nX1 := nX1.Value,
    nY1 := nY1.Value,
    nX2 := nX2.Value,
	nY2 := nY2.Value,
	ipDestImage := ipDestImage.Value,
    aColor := aColor.Value,
    nThickness := nThickness.Value,
	hrPrev:= hrPrev.Value);
END_METHOD

METHOD PUBLIC PreExecutionCheck
VAR_INPUT
	Check : I_PreExecutionChecks;
END_VAR
Check.IsTrue(ipDestImage.IsValid, 'ipDestImage must contain an image');
Check.IsTrue(nThickness.Value >= 1, 'nThickness must be greater than or equal to 1');
END_METHOD

END_FUNCTION_BLOCK

// Nodes/Drawing/Node_F_VN_DrawLine_TcVnVector4_DINT
{attribute 'linkalways'} 
{attribute 'no_explicit_call' := 'This FB is a CLASS and must be accessed using methods or properties'}
{attribute 'enable_dynamic_creation'}
FUNCTION_BLOCK Node_F_VN_DrawLine_TcVnVector4_DINT EXTENDS VisionNode
VAR
    aLine : _TcVnVector4_DINT;
    ipDestImage : _ITcVnImage;
    aColor : _TcVnVector4_LREAL;
    nThickness : _DINT(1);
    hrPrev : _HRESULT(S_OK);
	hresult : _HRESULT(S_OK);
END_VAR

METHOD FB_init : BOOL
VAR_INPUT
	bInitRetains : BOOL; // if TRUE, the retain variables are initialized (warm start / cold start)
	bInCopyCode : BOOL;  // if TRUE, the instance afterwards gets moved into the copy code (online change)
END_VAR
AddInput('aLine', aLine);
AddInput('ipDestImage', ipDestImage);
AddInput('aColor', aColor);
AddInput('hrPrev', hrPrev);
AddOutput('ipDestImage', ipDestImage);
AddOutput('hresult',hresult);
AddParameter('nThickness', nThickness);
END_METHOD

METHOD PUBLIC  Clone : I_Node
VAR
	pNode : POINTER TO Node_F_VN_DrawLine_TcVnVector4_DINT;
END_VAR
pNode := __NEW(Node_F_VN_DrawLine_TcVnVector4_DINT);
Clone := pNode^;
END_METHOD

METHOD PROTECTED OnExecute
hresult.Value := F_VN_DrawLine_TcVnVector4_DINT(
    aLine := aLine.Value,
	ipDestImage := ipDestImage.Value,
    aColor := aColor.Value,
    nThickness := nThickness.Value,
	hrPrev:= hrPrev.Value);
END_METHOD

METHOD PUBLIC PreExecutionCheck
VAR_INPUT
	Check : I_PreExecutionChecks;
END_VAR
Check.IsTrue(ipDestImage.IsValid, 'ipDestImage must contain an image');
Check.IsTrue(nThickness.Value >= 1, 'nThickness must be greater than or equal to 1');
END_METHOD

END_FUNCTION_BLOCK

// Nodes/Drawing/Node_F_VN_DrawLine_TcVnVector4_LREAL
{attribute 'linkalways'} 
{attribute 'no_explicit_call' := 'This FB is a CLASS and must be accessed using methods or properties'}
{attribute 'enable_dynamic_creation'}
FUNCTION_BLOCK Node_F_VN_DrawLine_TcVnVector4_LREAL EXTENDS VisionNode
VAR
    aLine : _TcVnVector4_LREAL;
    ipDestImage : _ITcVnImage;
    aColor : _TcVnVector4_LREAL;
    nThickness : _DINT(1);
    hrPrev : _HRESULT(S_OK);
	hresult : _HRESULT(S_OK);
END_VAR

METHOD FB_init : BOOL
VAR_INPUT
	bInitRetains : BOOL; // if TRUE, the retain variables are initialized (warm start / cold start)
	bInCopyCode : BOOL;  // if TRUE, the instance afterwards gets moved into the copy code (online change)
END_VAR
AddInput('aLine', aLine);
AddInput('ipDestImage', ipDestImage);
AddInput('aColor', aColor);
AddInput('hrPrev', hrPrev);
AddOutput('ipDestImage', ipDestImage);
AddOutput('hresult',hresult);
AddParameter('nThickness', nThickness);
END_METHOD

METHOD PUBLIC  Clone : I_Node
VAR
	pNode : POINTER TO Node_F_VN_DrawLine_TcVnVector4_LREAL;
END_VAR
pNode := __NEW(Node_F_VN_DrawLine_TcVnVector4_LREAL);
Clone := pNode^;
END_METHOD

METHOD PROTECTED OnExecute
hresult.Value := F_VN_DrawLine_TcVnVector4_LREAL(
    aLine := aLine.Value,
	ipDestImage := ipDestImage.Value,
    aColor := aColor.Value,
    nThickness := nThickness.Value,
	hrPrev:= hrPrev.Value);
END_METHOD

METHOD PUBLIC PreExecutionCheck
VAR_INPUT
	Check : I_PreExecutionChecks;
END_VAR
Check.IsTrue(ipDestImage.IsValid, 'ipDestImage must contain an image');
Check.IsTrue(nThickness.Value >= 1, 'nThickness must be greater than or equal to 1');
END_METHOD

END_FUNCTION_BLOCK

// Nodes/Drawing/Node_F_VN_DrawLineExp
{attribute 'linkalways'} 
{attribute 'no_explicit_call' := 'This FB is a CLASS and must be accessed using methods or properties'}
{attribute 'enable_dynamic_creation'}
FUNCTION_BLOCK Node_F_VN_DrawLineExp EXTENDS VisionNode
VAR
    nX1 : _UDINT(0);
    nY1 : _UDINT(0);
    nX2 : _UDINT(0);
    nY2 : _UDINT(0);
    ipDestImage : _ITcVnImage;
    aColor : _TcVnVector4_LREAL;
    nThickness : _DINT(1);
    eLineType : _ETcVnLineType(ETcVnLineType.TCVN_LT_4_CONNECTED);
    nShift : _UDINT(0);
    hrPrev : _HRESULT(S_OK);
	hresult : _HRESULT(S_OK);
END_VAR

METHOD FB_init : BOOL
VAR_INPUT
	bInitRetains : BOOL; // if TRUE, the retain variables are initialized (warm start / cold start)
	bInCopyCode : BOOL;  // if TRUE, the instance afterwards gets moved into the copy code (online change)
END_VAR
AddParameter('nX1', nX1);
AddParameter('nY1', nY1);
AddParameter('nX2', nX2);
AddParameter('nY2', nY2);
AddInput('ipDestImage', ipDestImage);
AddInput('aColor', aColor);
AddParameter('nThickness', nThickness);
AddParameter('eLineType', eLineType);
AddParameter('nShift', nShift);
AddInput('hrPrev', hrPrev);
AddOutput('ipDestImage', ipDestImage);
AddOutput('hresult',hresult);
END_METHOD

METHOD PUBLIC  Clone : I_Node
VAR
	pNode : POINTER TO Node_F_VN_DrawLineExp;
END_VAR
pNode := __NEW(Node_F_VN_DrawLineExp);
Clone := pNode^;
END_METHOD

METHOD PROTECTED OnExecute
hresult.Value := F_VN_DrawLineExp(
    nX1 := nX1.Value,
    nY1 := nY1.Value,
    nX2 := nX2.Value,
	nY2 := nY2.Value,
	ipDestImage := ipDestImage.Value,
    aColor := aColor.Value,
    nThickness := nThickness.Value,
    eLineType := eLineType.Value,
    nShift := nShift.Value,
	hrPrev:= hrPrev.Value);
END_METHOD

METHOD PUBLIC PreExecutionCheck
VAR_INPUT
	Check : I_PreExecutionChecks;
END_VAR
Check.IsTrue(ipDestImage.IsValid, 'ipDestImage must contain an image');
Check.IsTrue(nThickness.Value >= 1, 'nThickness must be greater than or equal to 1');
END_METHOD

END_FUNCTION_BLOCK

// Nodes/Drawing/Node_F_VN_DrawLineExp_TcVnVector4_DINT
{attribute 'linkalways'} 
{attribute 'no_explicit_call' := 'This FB is a CLASS and must be accessed using methods or properties'}
{attribute 'enable_dynamic_creation'}
FUNCTION_BLOCK Node_F_VN_DrawLineExp_TcVnVector4_DINT EXTENDS VisionNode
VAR
    aLine : _TcVnVector4_DINT;
    ipDestImage : _ITcVnImage;
    aColor : _TcVnVector4_LREAL;
    nThickness : _DINT(1);
    eLineType : _ETcVnLineType(ETcVnLineType.TCVN_LT_4_CONNECTED);
    nShift : _UDINT(0);
    hrPrev : _HRESULT(S_OK);
	hresult : _HRESULT(S_OK);
END_VAR

METHOD FB_init : BOOL
VAR_INPUT
	bInitRetains : BOOL; // if TRUE, the retain variables are initialized (warm start / cold start)
	bInCopyCode : BOOL;  // if TRUE, the instance afterwards gets moved into the copy code (online change)
END_VAR
AddInput('aLine', aLine);
AddInput('ipDestImage', ipDestImage);
AddInput('aColor', aColor);
AddParameter('nThickness', nThickness);
AddParameter('eLineType', eLineType);
AddParameter('nShift', nShift);
AddInput('hrPrev', hrPrev);
AddOutput('ipDestImage', ipDestImage);
AddOutput('hresult',hresult);
END_METHOD

METHOD PUBLIC  Clone : I_Node
VAR
	pNode : POINTER TO Node_F_VN_DrawLineExp_TcVnVector4_DINT;
END_VAR
pNode := __NEW(Node_F_VN_DrawLineExp_TcVnVector4_DINT);
Clone := pNode^;
END_METHOD

METHOD PROTECTED OnExecute
hresult.Value := F_VN_DrawLineExp_TcVnVector4_DINT(
    aLine := aLine.Value,
	ipDestImage := ipDestImage.Value,
    aColor := aColor.Value,
    nThickness := nThickness.Value,
    eLineType := eLineType.Value,
    nShift := nShift.Value,
	hrPrev:= hrPrev.Value);
END_METHOD

METHOD PUBLIC PreExecutionCheck
VAR_INPUT
	Check : I_PreExecutionChecks;
END_VAR
Check.IsTrue(ipDestImage.IsValid, 'ipDestImage must contain an image');
Check.IsTrue(nThickness.Value >= 1, 'nThickness must be greater than or equal to 1');
END_METHOD

END_FUNCTION_BLOCK

// Nodes/Drawing/Node_F_VN_DrawLineExp_TcVnVector4_LREAL
{attribute 'linkalways'} 
{attribute 'no_explicit_call' := 'This FB is a CLASS and must be accessed using methods or properties'}
{attribute 'enable_dynamic_creation'}
FUNCTION_BLOCK Node_F_VN_DrawLineExp_TcVnVector4_LREAL EXTENDS VisionNode
VAR
    aLine : _TcVnVector4_LREAL;
    ipDestImage : _ITcVnImage;
    aColor : _TcVnVector4_LREAL;
    nThickness : _DINT(1);
    eLineType : _ETcVnLineType(ETcVnLineType.TCVN_LT_4_CONNECTED);
    nShift : _UDINT(0);
    hrPrev : _HRESULT(S_OK);
	hresult : _HRESULT(S_OK);
END_VAR

METHOD FB_init : BOOL
VAR_INPUT
	bInitRetains : BOOL; // if TRUE, the retain variables are initialized (warm start / cold start)
	bInCopyCode : BOOL;  // if TRUE, the instance afterwards gets moved into the copy code (online change)
END_VAR
AddInput('aLine', aLine);
AddInput('ipDestImage', ipDestImage);
AddInput('aColor', aColor);
AddParameter('nThickness', nThickness);
AddParameter('eLineType', eLineType);
AddParameter('nShift', nShift);
AddInput('hrPrev', hrPrev);
AddOutput('ipDestImage', ipDestImage);
AddOutput('hresult',hresult);
END_METHOD

METHOD PUBLIC  Clone : I_Node
VAR
	pNode : POINTER TO Node_F_VN_DrawLineExp_TcVnVector4_LREAL;
END_VAR
pNode := __NEW(Node_F_VN_DrawLineExp_TcVnVector4_LREAL);
Clone := pNode^;
END_METHOD

METHOD PROTECTED OnExecute
hresult.Value := F_VN_DrawLineExp_TcVnVector4_LREAL(
    aLine := aLine.Value,
	ipDestImage := ipDestImage.Value,
    aColor := aColor.Value,
    nThickness := nThickness.Value,
    eLineType := eLineType.Value,
    nShift := nShift.Value,
	hrPrev:= hrPrev.Value);
END_METHOD

METHOD PUBLIC PreExecutionCheck
VAR_INPUT
	Check : I_PreExecutionChecks;
END_VAR
Check.IsTrue(ipDestImage.IsValid, 'ipDestImage must contain an image');
Check.IsTrue(nThickness.Value >= 1, 'nThickness must be greater than or equal to 1');
END_METHOD

END_FUNCTION_BLOCK

// Nodes/Drawing/Node_F_VN_DrawLines
{attribute 'linkalways'} 
{attribute 'no_explicit_call' := 'This FB is a CLASS and must be accessed using methods or properties'}
{attribute 'enable_dynamic_creation'}
FUNCTION_BLOCK Node_F_VN_DrawLines EXTENDS VisionNode
VAR
    ipLines : _ITcVnContainer;
    nLineIndex : _DINT(0);
    ipDestImage : _ITcVnImage;
    aColor : _TcVnVector4_LREAL;
    nThickness : _DINT(1);
    hrPrev : _HRESULT(S_OK);
	hresult : _HRESULT(S_OK);
END_VAR

METHOD FB_init : BOOL
VAR_INPUT
	bInitRetains : BOOL; // if TRUE, the retain variables are initialized (warm start / cold start)
	bInCopyCode : BOOL;  // if TRUE, the instance afterwards gets moved into the copy code (online change)
END_VAR
AddInput('ipLines', ipLines);
AddParameter('nLineIndex', nLineIndex);
AddInput('ipDestImage', ipDestImage);
AddInput('aColor', aColor);
AddParameter('nThickness', nThickness);
AddInput('hrPrev', hrPrev);
AddOutput('ipDestImage', ipDestImage);
AddOutput('hresult',hresult);
END_METHOD

METHOD PUBLIC  Clone : I_Node
VAR
	pNode : POINTER TO Node_F_VN_DrawLines;
END_VAR
pNode := __NEW(Node_F_VN_DrawLines);
Clone := pNode^;
END_METHOD

METHOD PROTECTED OnExecute
hresult.Value := F_VN_DrawLines(
    ipLines := ipLines.Value,
    nLineIndex := nLineIndex.Value,
	ipDestImage := ipDestImage.Value,
    aColor := aColor.Value,
    nThickness := nThickness.Value,
	hrPrev:= hrPrev.Value);
END_METHOD

METHOD PUBLIC PreExecutionCheck
VAR_INPUT
	Check : I_PreExecutionChecks;
END_VAR
Check.IsTrue(ipLines.IsValid, 'ipLines must be a valid container');

Check.IsTrue((ipLines.IsType(TC_GLOBAL_CONST_LIST.ContainerType_Vector_TcVnVector2_REAL) OR
              ipLines.IsType(TC_GLOBAL_CONST_LIST.ContainerType_Vector_TcVnVector4_LREAL) OR
              ipLines.IsType(TC_GLOBAL_CONST_LIST.ContainerType_Vector_TcVnVector4_DINT)),
              'ipLines contains incorrect type');
              
Check.IsTrue(ipDestImage.IsValid, 'ipDestImage must contain an image');
Check.IsTrue(nThickness.Value >= 1, 'nThickness must be greater than or equal to 1');
END_METHOD

END_FUNCTION_BLOCK

// Nodes/Drawing/Node_F_VN_DrawLinesExp
{attribute 'linkalways'} 
{attribute 'no_explicit_call' := 'This FB is a CLASS and must be accessed using methods or properties'}
{attribute 'enable_dynamic_creation'}
FUNCTION_BLOCK Node_F_VN_DrawLinesExp EXTENDS VisionNode
VAR
    ipLines : _ITcVnContainer;
    nLineIndex : _DINT(0);
    ipDestImage : _ITcVnImage;
    aColor : _TcVnVector4_LREAL;
    nThickness : _DINT(1);
    eLineType : _ETcVnLineType(ETcVnLineType.TCVN_LT_4_CONNECTED);
    nShift : _UDINT(0);
    hrPrev : _HRESULT(S_OK);
	hresult : _HRESULT(S_OK);
END_VAR

METHOD FB_init : BOOL
VAR_INPUT
	bInitRetains : BOOL; // if TRUE, the retain variables are initialized (warm start / cold start)
	bInCopyCode : BOOL;  // if TRUE, the instance afterwards gets moved into the copy code (online change)
END_VAR
AddInput('ipLines', ipLines);
AddParameter('nLineIndex', nLineIndex);
AddInput('ipDestImage', ipDestImage);
AddInput('aColor', aColor);
AddParameter('nThickness', nThickness);
AddParameter('eLineType', eLineType);
AddParameter('nShift', nShift);
AddInput('hrPrev', hrPrev);
AddOutput('ipDestImage', ipDestImage);
AddOutput('hresult',hresult);
END_METHOD

METHOD PUBLIC  Clone : I_Node
VAR
	pNode : POINTER TO Node_F_VN_DrawLinesExp;
END_VAR
pNode := __NEW(Node_F_VN_DrawLinesExp);
Clone := pNode^;
END_METHOD

METHOD PROTECTED OnExecute
hresult.Value := F_VN_DrawLinesExp(
    ipLines := ipLines.Value,
    nLineIndex := nLineIndex.Value,
	ipDestImage := ipDestImage.Value,
    aColor := aColor.Value,
    nThickness := nThickness.Value,
    eLineType := eLineType.Value,
    nShift := nShift.Value,
	hrPrev:= hrPrev.Value);
END_METHOD

METHOD PUBLIC PreExecutionCheck
VAR_INPUT
	Check : I_PreExecutionChecks;
END_VAR
Check.IsTrue(ipLines.IsValid, 'ipLines must be a valid container');

Check.IsTrue((ipLines.IsType(TC_GLOBAL_CONST_LIST.ContainerType_Vector_TcVnVector2_REAL) OR
              ipLines.IsType(TC_GLOBAL_CONST_LIST.ContainerType_Vector_TcVnVector4_LREAL) OR
              ipLines.IsType(TC_GLOBAL_CONST_LIST.ContainerType_Vector_TcVnVector4_DINT)),
              'ipLines contains incorrect type');
              
Check.IsTrue(ipDestImage.IsValid, 'ipDestImage must contain an image');
Check.IsTrue(nThickness.Value >= 1, 'nThickness must be greater than or equal to 1');
END_METHOD

END_FUNCTION_BLOCK

// Nodes/Drawing/Node_F_VN_DrawMatches
{attribute 'linkalways'} 
{attribute 'no_explicit_call' := 'This FB is a CLASS and must be accessed using methods or properties'}
{attribute 'enable_dynamic_creation'}
FUNCTION_BLOCK Node_F_VN_DrawMatches EXTENDS VisionNode
VAR
    ipSrcImage1 : _ITcVnImage;
    ipKeyPoints1 : _ITcVnContainer;
    ipSrcImage2 : _ITcVnImage;
    ipKeyPoints2 : _ITcVnContainer;
    ipMatches1To2 : _ITcVnContainer;
    ipDestImage : _ITcVnImage;
    hrPrev : _HRESULT(S_OK);
	hresult : _HRESULT(S_OK);
END_VAR

METHOD FB_init : BOOL
VAR_INPUT
	bInitRetains : BOOL; // if TRUE, the retain variables are initialized (warm start / cold start)
	bInCopyCode : BOOL;  // if TRUE, the instance afterwards gets moved into the copy code (online change)
END_VAR
AddInput('ipSrcImage1', ipSrcImage1);
AddInput('ipKeyPoints1', ipKeyPoints1);
AddInput('ipSrcImage2', ipSrcImage2);
AddInput('ipKeyPoints2', ipKeyPoints2);
AddInput('ipMatches1To2', ipMatches1To2);
AddInput('hrPrev', hrPrev);
AddOutput('ipDestImage', ipDestImage);
AddOutput('hresult',hresult);
END_METHOD

METHOD PUBLIC  Clone : I_Node
VAR
	pNode : POINTER TO Node_F_VN_DrawMatches
;
END_VAR
pNode := __NEW(Node_F_VN_DrawMatches);
Clone := pNode^;
END_METHOD

METHOD PROTECTED OnExecute
hresult.Value := F_VN_DrawMatches(
    ipSrcImage1 := ipSrcImage1.Value,
    ipKeyPoints1 := ipKeyPoints1.Value,
    ipSrcImage2 := ipSrcImage2.Value,
    ipKeyPoints2 := ipKeyPoints2.Value,
    ipMatches1To2 := ipMatches1To2.Value,
	ipDestImage := ipDestImage.Value,
	hrPrev:= hrPrev.Value);
END_METHOD

METHOD PUBLIC PreExecutionCheck
VAR_INPUT
	Check : I_PreExecutionChecks;
END_VAR
VAR
    srcImage1PixelFormat : TcVnPixelFormat;
    srcImage2PixelFormat : TcVnPixelFormat;
END_VAR
Check.IsTrue(ipSrcImage1.IsValid, 'ipSrcImage1 must contain an image');
Check.IsTrue(ipSrcImage1.IsPixelDepth(8), 'ipSrcImage1 must have 8 bit pixel depth');
Check.IsTrue(ipSrcImage1.TryGetPixelFormat(srcImage1PixelFormat), 'Failed to get ipSrcImage1 pixel format');

Check.IsTrue(ipSrcImage2.IsValid, 'ipSrcImage2 must contain an image');
Check.IsTrue(ipSrcImage2.IsPixelDepth(8), 'ipSrcImage2 must have 8 bit pixel depth');
Check.IsTrue(ipSrcImage2.TryGetPixelFormat(srcImage2PixelFormat), 'Failed to get ipSrcImage2 pixel format');

Check.IsTrue((srcImage1PixelFormat.nChannels = srcImage2PixelFormat.nChannels), 'ipSrcImage2 must have same number of channels as ipSrcImage1');

Check.IsTrue(ipKeyPoints1.IsType(TC_GLOBAL_CONST_LIST.ContainerType_Vector_TcVnKeyPoint), 'ipKeyPoints1 contains incorrect type');
Check.IsTrue(ipKeyPoints2.IsType(TC_GLOBAL_CONST_LIST.ContainerType_Vector_TcVnKeyPoint), 'ipKeyPoints2 contains incorrect type');
Check.IsTrue(ipMatches1To2.IsType(TC_GLOBAL_CONST_LIST.ContainerType_Vector_TcVnDMatch), 'ipMatches1To2 contains incorrect type');
END_METHOD

END_FUNCTION_BLOCK

// Nodes/Drawing/Node_F_VN_DrawMatchesExp
{attribute 'linkalways'} 
{attribute 'no_explicit_call' := 'This FB is a CLASS and must be accessed using methods or properties'}
{attribute 'enable_dynamic_creation'}
FUNCTION_BLOCK Node_F_VN_DrawMatchesExp EXTENDS VisionNode
VAR
    ipSrcImage1 : _ITcVnImage;
    ipKeyPoints1 : _ITcVnContainer;
    ipSrcImage2 : _ITcVnImage;
    ipKeyPoints2 : _ITcVnContainer;
    ipMatches1To2 : _ITcVnContainer;
    ipDestImage : _ITcVnImage;
    aMatchColor : _TcVnVector4_LREAL;
    aSingleColor : _TcVnVector4_LREAL;
    ipMatchesMask : _ITcVnContainer;
    eFlags : _ETcVnDrawMatchesFlags(ETcVnDrawMatchesFlags.TCVN_DMF_DEFAULT);
    hrPrev : _HRESULT(S_OK);
	hresult : _HRESULT(S_OK);
END_VAR

METHOD FB_init : BOOL
VAR_INPUT
	bInitRetains : BOOL; // if TRUE, the retain variables are initialized (warm start / cold start)
	bInCopyCode : BOOL;  // if TRUE, the instance afterwards gets moved into the copy code (online change)
END_VAR
AddInput('ipSrcImage1', ipSrcImage1);
AddInput('ipKeyPoints1', ipKeyPoints1);
AddInput('ipSrcImage2', ipSrcImage2);
AddInput('ipKeyPoints2', ipKeyPoints2);
AddInput('ipMatches1To2', ipMatches1To2);
AddInput('aMatchColor', aMatchColor);
AddInput('aSingleColor', aSingleColor);
AddInput('ipMatchesMask', ipMatchesMask);
AddParameter('eFlags', eFlags);
AddInput('hrPrev', hrPrev);
AddOutput('ipDestImage', ipDestImage);
AddOutput('hresult',hresult);
END_METHOD

METHOD PUBLIC  Clone : I_Node
VAR
	pNode : POINTER TO Node_F_VN_DrawMatchesExp
;
END_VAR
pNode := __NEW(Node_F_VN_DrawMatchesExp);
Clone := pNode^;
END_METHOD

METHOD PROTECTED OnExecute
hresult.Value := F_VN_DrawMatchesExp(
    ipSrcImage1 := ipSrcImage1.Value,
    ipKeyPoints1 := ipKeyPoints1.Value,
    ipSrcImage2 := ipSrcImage2.Value,
    ipKeyPoints2 := ipKeyPoints2.Value,
    ipMatches1To2 := ipMatches1To2.Value,
	ipDestImage := ipDestImage.Value,
    aMatchColor := aMatchColor.Value,
    aSingleColor := aSingleColor.Value,
    ipMatchesMask := ipMatchesMask.Value,
    eFlags := eFlags.Value,
	hrPrev:= hrPrev.Value);
END_METHOD

METHOD PUBLIC PreExecutionCheck
VAR_INPUT
	Check : I_PreExecutionChecks;
END_VAR
VAR
    srcImage1PixelFormat : TcVnPixelFormat;
    srcImage2PixelFormat : TcVnPixelFormat;
END_VAR
Check.IsTrue(ipSrcImage1.IsValid, 'ipSrcImage1 must contain an image');
Check.IsTrue(ipSrcImage1.IsPixelDepth(8), 'ipSrcImage1 must have 8 bit pixel depth');
Check.IsTrue(ipSrcImage1.TryGetPixelFormat(srcImage1PixelFormat), 'Failed to get ipSrcImage1 pixel format');

Check.IsTrue(ipSrcImage2.IsValid, 'ipSrcImage2 must contain an image');
Check.IsTrue(ipSrcImage2.IsPixelDepth(8), 'ipSrcImage2 must have 8 bit pixel depth');
Check.IsTrue(ipSrcImage2.TryGetPixelFormat(srcImage2PixelFormat), 'Failed to get ipSrcImage2 pixel format');

Check.IsTrue((srcImage1PixelFormat.nChannels = srcImage2PixelFormat.nChannels), 'ipSrcImage2 must have same number of channels as ipSrcImage1');

Check.IsTrue(ipKeyPoints1.IsType(TC_GLOBAL_CONST_LIST.ContainerType_Vector_TcVnKeyPoint), 'ipKeyPoints1 contains incorrect type');
Check.IsTrue(ipKeyPoints2.IsType(TC_GLOBAL_CONST_LIST.ContainerType_Vector_TcVnKeyPoint), 'ipKeyPoints2 contains incorrect type');
Check.IsTrue(ipMatches1To2.IsType(TC_GLOBAL_CONST_LIST.ContainerType_Vector_TcVnDMatch), 'ipMatches1To2 contains incorrect type');

IF ipMatchesMask.IsValid THEN
    Check.IsTrue(ipMatchesMask.IsType(TC_GLOBAL_CONST_LIST.ContainerType_Vector_SINT), 'ipMatchesMask contains incorrect type');
END_IF
END_METHOD

END_FUNCTION_BLOCK

// Nodes/Drawing/Node_F_VN_DrawOrientation
{attribute 'linkalways'} 
{attribute 'no_explicit_call' := 'This FB is a CLASS and must be accessed using methods or properties'}
{attribute 'enable_dynamic_creation'}
FUNCTION_BLOCK Node_F_VN_DrawOrientation EXTENDS VisionNode
VAR
    stOrientation : _TcVnRotatedRectangle;
    ipDestImage : _ITcVnImage;
    aColorMainAxis : _TcVnVector4_LREAL;
    nThickness : _DINT(1);
    hrPrev : _HRESULT(S_OK);
	hresult : _HRESULT(S_OK);
END_VAR

METHOD FB_init : BOOL
VAR_INPUT
	bInitRetains : BOOL; // if TRUE, the retain variables are initialized (warm start / cold start)
	bInCopyCode : BOOL;  // if TRUE, the instance afterwards gets moved into the copy code (online change)
END_VAR
AddInput('stOrientation', stOrientation);
AddInput('ipDestImage', ipDestImage);
AddInput('aColorMainAxis', aColorMainAxis);
AddParameter('nThickness', nThickness);
AddInput('hrPrev', hrPrev);
AddOutput('ipDestImage', ipDestImage);
AddOutput('hresult',hresult);
END_METHOD

METHOD PUBLIC  Clone : I_Node
VAR
	pNode : POINTER TO Node_F_VN_DrawOrientation;
END_VAR
pNode := __NEW(Node_F_VN_DrawOrientation);
Clone := pNode^;
END_METHOD

METHOD PROTECTED OnExecute
hresult.Value := F_VN_DrawOrientation(
    stOrientation := stOrientation.Value,
	ipDestImage := ipDestImage.Value,
    aColorMainAxis := aColorMainAxis.Value,
    nThickness := nThickness.Value,
	hrPrev:= hrPrev.Value);
END_METHOD

METHOD PUBLIC PreExecutionCheck
VAR_INPUT
	Check : I_PreExecutionChecks;
END_VAR
Check.IsTrue(ipDestImage.IsValid, 'ipDestImage must contain an image');
Check.IsTrue(nThickness.Value >= 1, 'nThickness must be greater than or equal to 1');
END_METHOD

END_FUNCTION_BLOCK

// Nodes/Drawing/Node_F_VN_DrawOrientationExp
{attribute 'linkalways'} 
{attribute 'no_explicit_call' := 'This FB is a CLASS and must be accessed using methods or properties'}
{attribute 'enable_dynamic_creation'}
FUNCTION_BLOCK Node_F_VN_DrawOrientationExp EXTENDS VisionNode
VAR
    stOrientation : _TcVnRotatedRectangle;
    ipDestImage : _ITcVnImage;
    aColorMainAxis : _TcVnVector4_LREAL;
    nThickness : _DINT(1);
    aColorHorizontalAxis : _TcVnVector4_LREAL;
    fFontScale : _LREAL(1.0);
    hrPrev : _HRESULT(S_OK);
	hresult : _HRESULT(S_OK);
END_VAR

METHOD FB_init : BOOL
VAR_INPUT
	bInitRetains : BOOL; // if TRUE, the retain variables are initialized (warm start / cold start)
	bInCopyCode : BOOL;  // if TRUE, the instance afterwards gets moved into the copy code (online change)
END_VAR
AddInput('stOrientation', stOrientation);
AddInput('ipDestImage', ipDestImage);
AddInput('aColorMainAxis', aColorMainAxis);
AddParameter('nThickness', nThickness);
AddInput('aColorHorizontalAxis', aColorHorizontalAxis);
AddParameter('fFontScale', fFontScale);
AddInput('hrPrev', hrPrev);
AddOutput('ipDestImage', ipDestImage);
AddOutput('hresult',hresult);
END_METHOD

METHOD PUBLIC  Clone : I_Node
VAR
	pNode : POINTER TO Node_F_VN_DrawOrientationExp;
END_VAR
pNode := __NEW(Node_F_VN_DrawOrientationExp);
Clone := pNode^;
END_METHOD

METHOD PROTECTED OnExecute
hresult.Value := F_VN_DrawOrientationExp(
    stOrientation := stOrientation.Value,
	ipDestImage := ipDestImage.Value,
    aColorMainAxis := aColorMainAxis.Value,
    nThickness := nThickness.Value,
    aColorHorizontalAxis := aColorHorizontalAxis.Value,
    fFontScale := fFontScale.Value,
	hrPrev:= hrPrev.Value);
END_METHOD

METHOD PUBLIC PreExecutionCheck
VAR_INPUT
	Check : I_PreExecutionChecks;
END_VAR
Check.IsTrue(ipDestImage.IsValid, 'ipDestImage must contain an image');
Check.IsTrue(nThickness.Value >= 1, 'nThickness must be greater than or equal to 1');
END_METHOD

END_FUNCTION_BLOCK

// Nodes/Drawing/Node_F_VN_DrawPoint
{attribute 'linkalways'} 
{attribute 'no_explicit_call' := 'This FB is a CLASS and must be accessed using methods or properties'}
{attribute 'enable_dynamic_creation'}
FUNCTION_BLOCK Node_F_VN_DrawPoint EXTENDS VisionNode
VAR
    nX : _UDINT(0);
    nY : _UDINT(0);
    ipDestImage : _ITcVnImage;
    eShape : _ETcVnDrawShape(ETcVnDrawShape.TCVN_DS_CIRCLE);
    aColor : _TcVnVector4_LREAL;
    hrPrev : _HRESULT(S_OK);
	hresult : _HRESULT(S_OK);
END_VAR

METHOD FB_init : BOOL
VAR_INPUT
	bInitRetains : BOOL; // if TRUE, the retain variables are initialized (warm start / cold start)
	bInCopyCode : BOOL;  // if TRUE, the instance afterwards gets moved into the copy code (online change)
END_VAR
AddParameter('nX', nX);
AddParameter('nY', nY);
AddInput('ipDestImage', ipDestImage);
AddParameter('eShape', eShape);
AddInput('aColor', aColor);
AddInput('hrPrev', hrPrev);
AddOutput('ipDestImage', ipDestImage);
AddOutput('hresult',hresult);
END_METHOD

METHOD PUBLIC  Clone : I_Node
VAR
	pNode : POINTER TO Node_F_VN_DrawPoint;
END_VAR
pNode := __NEW(Node_F_VN_DrawPoint);
Clone := pNode^;
END_METHOD

METHOD PROTECTED OnExecute
hresult.Value := F_VN_DrawPoint(
    nX := nX.Value,
    nY := nY.Value,
	ipDestImage := ipDestImage.Value,
    eShape := eShape.Value,
    aColor := aColor.Value,
	hrPrev:= hrPrev.Value);
END_METHOD

METHOD PUBLIC PreExecutionCheck
VAR_INPUT
	Check : I_PreExecutionChecks;
END_VAR
Check.IsTrue(ipDestImage.IsValid, 'ipDestImage must contain an image');
END_METHOD

END_FUNCTION_BLOCK

// Nodes/Drawing/Node_F_VN_DrawPointExp
{attribute 'linkalways'} 
{attribute 'no_explicit_call' := 'This FB is a CLASS and must be accessed using methods or properties'}
{attribute 'enable_dynamic_creation'}
FUNCTION_BLOCK Node_F_VN_DrawPointExp EXTENDS VisionNode
VAR
    nX : _UDINT(0);
    nY : _UDINT(0);
    ipDestImage : _ITcVnImage;
    eShape : _ETcVnDrawShape(ETcVnDrawShape.TCVN_DS_CIRCLE);
    aColor : _TcVnVector4_LREAL;
    nSize  : _UDINT(0);
    nThickness : _DINT(1);
    eLineType : _ETcVnLineType(ETcVnLineType.TCVN_LT_4_CONNECTED);
    hrPrev : _HRESULT(S_OK);
	hresult : _HRESULT(S_OK);
END_VAR

METHOD FB_init : BOOL
VAR_INPUT
	bInitRetains : BOOL; // if TRUE, the retain variables are initialized (warm start / cold start)
	bInCopyCode : BOOL;  // if TRUE, the instance afterwards gets moved into the copy code (online change)
END_VAR
AddParameter('nX', nX);
AddParameter('nY', nY);
AddInput('ipDestImage', ipDestImage);
AddParameter('eShape', eShape);
AddInput('aColor', aColor);
AddParameter('nSize', nSize);
AddParameter('nThickness', nThickness);
AddParameter('eLineType', eLineType);
AddInput('hrPrev', hrPrev);
AddOutput('ipDestImage', ipDestImage);
AddOutput('hresult',hresult);
END_METHOD

METHOD PUBLIC  Clone : I_Node
VAR
	pNode : POINTER TO Node_F_VN_DrawPointExp;
END_VAR
pNode := __NEW(Node_F_VN_DrawPointExp);
Clone := pNode^;
END_METHOD

METHOD PROTECTED OnExecute
hresult.Value := F_VN_DrawPointExp(
    nX := nX.Value,
    nY := nY.Value,
	ipDestImage := ipDestImage.Value,
    eShape := eShape.Value,
    aColor := aColor.Value,
    nSize := nSize.Value,
    nThickness := nThickness.Value,
    eLineType := eLineType.Value,
	hrPrev:= hrPrev.Value);
END_METHOD

METHOD PUBLIC PreExecutionCheck
VAR_INPUT
	Check : I_PreExecutionChecks;
END_VAR
Check.IsTrue(ipDestImage.IsValid, 'ipDestImage must contain an image');
Check.IsTrue(nThickness.Value <> 0, 'nThickness must be non-zero');
END_METHOD

END_FUNCTION_BLOCK

// Nodes/Drawing/Node_F_VN_DrawPoints
{attribute 'linkalways'} 
{attribute 'no_explicit_call' := 'This FB is a CLASS and must be accessed using methods or properties'}
{attribute 'enable_dynamic_creation'}
FUNCTION_BLOCK Node_F_VN_DrawPoints EXTENDS VisionNode
VAR
    ipPoints : _ITcVnContainer;
    ipDestImage : _ITcVnImage;
    eShape : _ETcVnDrawShape(ETcVnDrawShape.TCVN_DS_CIRCLE);
    aColor : _TcVnVector4_LREAL;
    hrPrev : _HRESULT(S_OK);
	hresult : _HRESULT(S_OK);
END_VAR

METHOD FB_init : BOOL
VAR_INPUT
	bInitRetains : BOOL; // if TRUE, the retain variables are initialized (warm start / cold start)
	bInCopyCode : BOOL;  // if TRUE, the instance afterwards gets moved into the copy code (online change)
END_VAR
AddInput('ipPoints', ipPoints);
AddInput('ipDestImage', ipDestImage);
AddParameter('eShape', eShape);
AddInput('aColor', aColor);
AddInput('hrPrev', hrPrev);
AddOutput('ipDestImage', ipDestImage);
AddOutput('hresult',hresult);
END_METHOD

METHOD PUBLIC  Clone : I_Node
VAR
	pNode : POINTER TO Node_F_VN_DrawPoints;
END_VAR
pNode := __NEW(Node_F_VN_DrawPoints);
Clone := pNode^;
END_METHOD

METHOD PROTECTED OnExecute
hresult.Value := F_VN_DrawPoints(
    ipPoints := ipPoints.Value,
	ipDestImage := ipDestImage.Value,
    eShape := eShape.Value,
    aColor := aColor.Value,
	hrPrev:= hrPrev.Value);
END_METHOD

METHOD PUBLIC PreExecutionCheck
VAR_INPUT
	Check : I_PreExecutionChecks;
END_VAR
Check.IsTrue(ipPoints.IsValid, 'ipPoints must be a valid container');
Check.IsTrue((ipPoints.IsType(TC_GLOBAL_CONST_LIST.ContainerType_Vector_TcVnPoint2_DINT) OR
              ipPoints.IsType(TC_GLOBAL_CONST_LIST.ContainerType_Vector_TcVnPoint2_REAL)),
              'ipPoints contains incorrect type');
              
Check.IsTrue(ipDestImage.IsValid, 'ipDestImage must contain an image');
END_METHOD

END_FUNCTION_BLOCK

// Nodes/Drawing/Node_F_VN_DrawPointsExp
{attribute 'linkalways'} 
{attribute 'no_explicit_call' := 'This FB is a CLASS and must be accessed using methods or properties'}
{attribute 'enable_dynamic_creation'}
FUNCTION_BLOCK Node_F_VN_DrawPointsExp EXTENDS VisionNode
VAR
    ipPoints : _ITcVnContainer;
    ipDestImage : _ITcVnImage;
    eShape : _ETcVnDrawShape(ETcVnDrawShape.TCVN_DS_CIRCLE);
    aColor : _TcVnVector4_LREAL;
    nSize  : _UDINT(0);
    nThickness : _DINT(1);
    eLineType : _ETcVnLineType(ETcVnLineType.TCVN_LT_4_CONNECTED);
    hrPrev : _HRESULT(S_OK);
	hresult : _HRESULT(S_OK);
END_VAR

METHOD FB_init : BOOL
VAR_INPUT
	bInitRetains : BOOL; // if TRUE, the retain variables are initialized (warm start / cold start)
	bInCopyCode : BOOL;  // if TRUE, the instance afterwards gets moved into the copy code (online change)
END_VAR
AddInput('ipPoints', ipPoints);
AddInput('ipDestImage', ipDestImage);
AddParameter('eShape', eShape);
AddInput('aColor', aColor);
AddParameter('nSize', nSize);
AddParameter('nThickness', nThickness);
AddParameter('eLineType', eLineType);
AddInput('hrPrev', hrPrev);
AddOutput('ipDestImage', ipDestImage);
AddOutput('hresult',hresult);
END_METHOD

METHOD PUBLIC  Clone : I_Node
VAR
	pNode : POINTER TO Node_F_VN_DrawPointsExp;
END_VAR
pNode := __NEW(Node_F_VN_DrawPointsExp);
Clone := pNode^;
END_METHOD

METHOD PROTECTED OnExecute
hresult.Value := F_VN_DrawPointsExp(
    ipPoints := ipPoints.Value,
	ipDestImage := ipDestImage.Value,
    eShape := eShape.Value,
    aColor := aColor.Value,
    nSize := nSize.Value,
    nThickness := nThickness.Value,
    eLineType := eLineType.Value,
	hrPrev:= hrPrev.Value);
END_METHOD

METHOD PUBLIC PreExecutionCheck
VAR_INPUT
	Check : I_PreExecutionChecks;
END_VAR
Check.IsTrue(ipPoints.IsValid, 'ipPoints must be a valid container');
Check.IsTrue((ipPoints.IsType(TC_GLOBAL_CONST_LIST.ContainerType_Vector_TcVnPoint2_DINT) OR
              ipPoints.IsType(TC_GLOBAL_CONST_LIST.ContainerType_Vector_TcVnPoint2_REAL)),
              'ipPoints contains incorrect type');
              
Check.IsTrue(ipDestImage.IsValid, 'ipDestImage must contain an image');
Check.IsTrue(nThickness.Value <> 0, 'nThickness must be non-zero');
END_METHOD

END_FUNCTION_BLOCK

// Nodes/Drawing/Node_F_VN_DrawPolygon
{attribute 'linkalways'} 
{attribute 'no_explicit_call' := 'This FB is a CLASS and must be accessed using methods or properties'}
{attribute 'enable_dynamic_creation'}
FUNCTION_BLOCK Node_F_VN_DrawPolygon EXTENDS VisionNode
VAR
    ipPoints : _ITcVnContainer;
    ipDestImage : _ITcVnImage;
    aColor : _TcVnVector4_LREAL;
    nThickness : _DINT(1);
    hrPrev : _HRESULT(S_OK);
	hresult : _HRESULT(S_OK);
END_VAR

METHOD FB_init : BOOL
VAR_INPUT
	bInitRetains : BOOL; // if TRUE, the retain variables are initialized (warm start / cold start)
	bInCopyCode : BOOL;  // if TRUE, the instance afterwards gets moved into the copy code (online change)
END_VAR
AddInput('ipPoints', ipPoints);
AddInput('ipDestImage', ipDestImage);
AddInput('aColor', aColor);
AddParameter('nThickness', nThickness);
AddInput('hrPrev', hrPrev);
AddOutput('ipDestImage', ipDestImage);
AddOutput('hresult',hresult);
END_METHOD

METHOD PUBLIC  Clone : I_Node
VAR
	pNode : POINTER TO Node_F_VN_DrawPolygon
;
END_VAR
pNode := __NEW(Node_F_VN_DrawPolygon);
Clone := pNode^;
END_METHOD

METHOD PROTECTED OnExecute
hresult.Value := F_VN_DrawPolygon(
    ipPoints := ipPoints.Value,
	ipDestImage := ipDestImage.Value,
    aColor := aColor.Value,
    nThickness := nThickness.Value,
	hrPrev:= hrPrev.Value);
END_METHOD

METHOD PUBLIC PreExecutionCheck
VAR_INPUT
	Check : I_PreExecutionChecks;
END_VAR
Check.IsTrue(ipPoints.IsValid, 'ipContours must be a valid container');
Check.IsTrue((ipPoints.IsType(TC_GLOBAL_CONST_LIST.ContainerType_Vector_TcVnPoint2_DINT) OR
              ipPoints.IsType(TC_GLOBAL_CONST_LIST.ContainerType_Vector_TcVnPoint2_REAL) OR
              ipPoints.IsType(TC_GLOBAL_CONST_LIST.ContainerType_Vector_TcVnPoint2_LREAL)),
              'ipPoints contains incorrect type');

Check.IsTrue(ipDestImage.IsValid, 'ipDestImage must contain an image');
Check.IsTrue(nThickness.Value <> 0, 'nThickness must be non-zero');
END_METHOD

END_FUNCTION_BLOCK

// Nodes/Drawing/Node_F_VN_DrawPolygonExp
{attribute 'linkalways'} 
{attribute 'no_explicit_call' := 'This FB is a CLASS and must be accessed using methods or properties'}
{attribute 'enable_dynamic_creation'}
FUNCTION_BLOCK Node_F_VN_DrawPolygonExp EXTENDS VisionNode
VAR
    ipPoints : _ITcVnContainer;
    ipDestImage : _ITcVnImage;
    aColor : _TcVnVector4_LREAL;
    nThickness : _DINT(1);
    bIsClosed : _BOOL(FALSE);
    eLineType : _ETcVnLineType(ETcVnLineType.TCVN_LT_4_CONNECTED);
    nShift : _UDINT(0);
    hrPrev : _HRESULT(S_OK);
	hresult : _HRESULT(S_OK);
END_VAR

METHOD FB_init : BOOL
VAR_INPUT
	bInitRetains : BOOL; // if TRUE, the retain variables are initialized (warm start / cold start)
	bInCopyCode : BOOL;  // if TRUE, the instance afterwards gets moved into the copy code (online change)
END_VAR
AddInput('ipPoints', ipPoints);
AddInput('ipDestImage', ipDestImage);
AddInput('aColor', aColor);
AddParameter('nThickness', nThickness);
AddParameter('bIsClosed', bIsClosed);
AddParameter('eLineType', eLineType);
AddParameter('nShift', nShift);
AddInput('hrPrev', hrPrev);
AddOutput('ipDestImage', ipDestImage);
AddOutput('hresult',hresult);
END_METHOD

METHOD PUBLIC  Clone : I_Node
VAR
	pNode : POINTER TO Node_F_VN_DrawPolygonExp
;
END_VAR
pNode := __NEW(Node_F_VN_DrawPolygonExp);
Clone := pNode^;
END_METHOD

METHOD PROTECTED OnExecute
hresult.Value := F_VN_DrawPolygonExp(
    ipPoints := ipPoints.Value,
	ipDestImage := ipDestImage.Value,
    aColor := aColor.Value,
    nThickness := nThickness.Value,
    bIsClosed := bIsClosed.Value,
    eLineType := eLineType.Value,
    nShift := nShift.Value,
	hrPrev:= hrPrev.Value);
END_METHOD

METHOD PUBLIC PreExecutionCheck
VAR_INPUT
	Check : I_PreExecutionChecks;
END_VAR
Check.IsTrue(ipPoints.IsValid, 'ipContours must be a valid container');
Check.IsTrue((ipPoints.IsType(TC_GLOBAL_CONST_LIST.ContainerType_Vector_TcVnPoint2_DINT) OR
              ipPoints.IsType(TC_GLOBAL_CONST_LIST.ContainerType_Vector_TcVnPoint2_REAL) OR
              ipPoints.IsType(TC_GLOBAL_CONST_LIST.ContainerType_Vector_TcVnPoint2_LREAL)),
              'ipPoints contains incorrect type');

Check.IsTrue(ipDestImage.IsValid, 'ipDestImage must contain an image');
Check.IsTrue(nThickness.Value <> 0, 'nThickness must be non-zero');
END_METHOD

END_FUNCTION_BLOCK

// Nodes/Drawing/Node_F_VN_DrawRectangle
{attribute 'linkalways'} 
{attribute 'no_explicit_call' := 'This FB is a CLASS and must be accessed using methods or properties'}
{attribute 'enable_dynamic_creation'}
FUNCTION_BLOCK Node_F_VN_DrawRectangle EXTENDS VisionNode
VAR
    nTopLeftX : _UDINT(0);
    nTopLeftY : _UDINT(0);
    nBottomRightX : _UDINT(0);
    nBottomRightY : _UDINT(0);
    ipDestImage : _ITcVnImage;
    aColor : _TcVnVector4_LREAL;
    nThickness : _DINT(1);
    hrPrev : _HRESULT(S_OK);
	hresult : _HRESULT(S_OK);
END_VAR

METHOD FB_init : BOOL
VAR_INPUT
	bInitRetains : BOOL; // if TRUE, the retain variables are initialized (warm start / cold start)
	bInCopyCode : BOOL;  // if TRUE, the instance afterwards gets moved into the copy code (online change)
END_VAR
AddParameter('nTopLeftX', nTopLeftX);
AddParameter('nTopLeftY', nTopLeftY);
AddParameter('nBottomRightX', nBottomRightX);
AddParameter('nBottomRightY', nBottomRightY);
AddInput('ipDestImage', ipDestImage);
AddInput('aColor', aColor);
AddParameter('nThickness', nThickness);
AddInput('hrPrev', hrPrev);
AddOutput('ipDestImage', ipDestImage);
AddOutput('hresult',hresult);
END_METHOD

METHOD PUBLIC  Clone : I_Node
VAR
	pNode : POINTER TO Node_F_VN_DrawRectangle;
END_VAR
pNode := __NEW(Node_F_VN_DrawRectangle);
Clone := pNode^;
END_METHOD

METHOD PROTECTED OnExecute
hresult.Value := F_VN_DrawRectangle(
    nTopLeftX := nTopLeftX.Value,
    nTopLeftY := nTopLeftY.Value,
    nBottomRightX := nBottomRightX.Value,
    nBottomRightY := nBottomRightY.Value,
	ipDestImage := ipDestImage.Value,
    aColor := aColor.Value,
    nThickness := nThickness.Value,
	hrPrev:= hrPrev.Value);
END_METHOD

METHOD PUBLIC PreExecutionCheck
VAR_INPUT
	Check : I_PreExecutionChecks;
END_VAR
Check.IsTrue(ipDestImage.IsValid, 'ipDestImage must contain an image');
Check.IsTrue(nThickness.Value <> 0, 'nThickness must be non-zero');
END_METHOD

END_FUNCTION_BLOCK

// Nodes/Drawing/Node_F_VN_DrawRectangle_TcVnRectangle_DINT
{attribute 'linkalways'} 
{attribute 'no_explicit_call' := 'This FB is a CLASS and must be accessed using methods or properties'}
{attribute 'enable_dynamic_creation'}
FUNCTION_BLOCK Node_F_VN_DrawRectangle_TcVnRectangle_DINT EXTENDS VisionNode
VAR
    stRectangle : _TcVnRectangle_DINT;
    ipDestImage : _ITcVnImage;
    aColor : _TcVnVector4_LREAL;
    nThickness : _DINT(1);
    hrPrev : _HRESULT(S_OK);
	hresult : _HRESULT(S_OK);
END_VAR

METHOD FB_init : BOOL
VAR_INPUT
	bInitRetains : BOOL; // if TRUE, the retain variables are initialized (warm start / cold start)
	bInCopyCode : BOOL;  // if TRUE, the instance afterwards gets moved into the copy code (online change)
END_VAR
AddInput('stRectangle', stRectangle);
AddInput('ipDestImage', ipDestImage);
AddInput('aColor', aColor);
AddParameter('nThickness', nThickness);
AddInput('hrPrev', hrPrev);
AddOutput('ipDestImage', ipDestImage);
AddOutput('hresult',hresult);
END_METHOD

METHOD PUBLIC  Clone : I_Node
VAR
	pNode : POINTER TO Node_F_VN_DrawRectangle_TcVnRectangle_DINT;
END_VAR
pNode := __NEW(Node_F_VN_DrawRectangle_TcVnRectangle_DINT);
Clone := pNode^;
END_METHOD

METHOD PROTECTED OnExecute
hresult.Value := F_VN_DrawRectangle_TcVnRectangle_DINT(
    stRectangle := stRectangle.Value,
	ipDestImage := ipDestImage.Value,
    aColor := aColor.Value,
    nThickness := nThickness.Value,
	hrPrev:= hrPrev.Value);
END_METHOD

METHOD PUBLIC PreExecutionCheck
VAR_INPUT
	Check : I_PreExecutionChecks;
END_VAR
Check.IsTrue(ipDestImage.IsValid, 'ipDestImage must contain an image');
Check.IsTrue(nThickness.Value <> 0, 'nThickness must be non-zero');
END_METHOD

END_FUNCTION_BLOCK

// Nodes/Drawing/Node_F_VN_DrawRectangle_TcVnRectangle_UDINT
{attribute 'linkalways'} 
{attribute 'no_explicit_call' := 'This FB is a CLASS and must be accessed using methods or properties'}
{attribute 'enable_dynamic_creation'}
FUNCTION_BLOCK Node_F_VN_DrawRectangle_TcVnRectangle_UDINT EXTENDS VisionNode
VAR
    stRectangle : _TcVnRectangle_UDINT;
    ipDestImage : _ITcVnImage;
    aColor : _TcVnVector4_LREAL;
    nThickness : _DINT(1);
    hrPrev : _HRESULT(S_OK);
	hresult : _HRESULT(S_OK);
END_VAR

METHOD FB_init : BOOL
VAR_INPUT
	bInitRetains : BOOL; // if TRUE, the retain variables are initialized (warm start / cold start)
	bInCopyCode : BOOL;  // if TRUE, the instance afterwards gets moved into the copy code (online change)
END_VAR
AddInput('stRectangle', stRectangle);
AddInput('ipDestImage', ipDestImage);
AddInput('aColor', aColor);
AddParameter('nThickness', nThickness);
AddInput('hrPrev', hrPrev);
AddOutput('ipDestImage', ipDestImage);
AddOutput('hresult',hresult);
END_METHOD

METHOD PUBLIC  Clone : I_Node
VAR
	pNode : POINTER TO Node_F_VN_DrawRectangle_TcVnRectangle_UDINT;
END_VAR
pNode := __NEW(Node_F_VN_DrawRectangle_TcVnRectangle_UDINT);
Clone := pNode^;
END_METHOD

METHOD PROTECTED OnExecute
hresult.Value := F_VN_DrawRectangle_TcVnRectangle_UDINT(
    stRectangle := stRectangle.Value,
	ipDestImage := ipDestImage.Value,
    aColor := aColor.Value,
    nThickness := nThickness.Value,
	hrPrev:= hrPrev.Value);
END_METHOD

METHOD PUBLIC PreExecutionCheck
VAR_INPUT
	Check : I_PreExecutionChecks;
END_VAR
Check.IsTrue(ipDestImage.IsValid, 'ipDestImage must contain an image');
Check.IsTrue(nThickness.Value <> 0, 'nThickness must be non-zero');
END_METHOD

END_FUNCTION_BLOCK

// Nodes/Drawing/Node_F_VN_DrawRotatedRectangle
{attribute 'linkalways'} 
{attribute 'no_explicit_call' := 'This FB is a CLASS and must be accessed using methods or properties'}
{attribute 'enable_dynamic_creation'}
FUNCTION_BLOCK Node_F_VN_DrawRotatedRectangle EXTENDS VisionNode
VAR
    stRectangle : _TcVnRotatedRectangle;
    ipDestImage : _ITcVnImage;
    aColor : _TcVnVector4_LREAL;
    nThickness : _DINT(1);
    hrPrev : _HRESULT(S_OK);
	hresult : _HRESULT(S_OK);
END_VAR

METHOD FB_init : BOOL
VAR_INPUT
	bInitRetains : BOOL; // if TRUE, the retain variables are initialized (warm start / cold start)
	bInCopyCode : BOOL;  // if TRUE, the instance afterwards gets moved into the copy code (online change)
END_VAR
AddInput('stRectangle', stRectangle);
AddInput('ipDestImage', ipDestImage);
AddInput('aColor', aColor);
AddParameter('nThickness', nThickness);
AddInput('hrPrev', hrPrev);
AddOutput('ipDestImage', ipDestImage);
AddOutput('hresult',hresult);
END_METHOD

METHOD PUBLIC  Clone : I_Node
VAR
	pNode : POINTER TO Node_F_VN_DrawRotatedRectangle;
END_VAR
pNode := __NEW(Node_F_VN_DrawRotatedRectangle);
Clone := pNode^;
END_METHOD

METHOD PROTECTED OnExecute
hresult.Value := F_VN_DrawRotatedRectangle(
    stRectangle := stRectangle.Value,
	ipDestImage := ipDestImage.Value,
    aColor := aColor.Value,
    nThickness := nThickness.Value,
	hrPrev:= hrPrev.Value);
END_METHOD

METHOD PUBLIC PreExecutionCheck
VAR_INPUT
	Check : I_PreExecutionChecks;
END_VAR
Check.IsTrue(ipDestImage.IsValid, 'ipDestImage must contain an image');
Check.IsTrue(nThickness.Value <> 0, 'nThickness must be non-zero');
END_METHOD

END_FUNCTION_BLOCK

// Nodes/Drawing/Node_F_VN_DrawRotatedRectangleExp
{attribute 'linkalways'} 
{attribute 'no_explicit_call' := 'This FB is a CLASS and must be accessed using methods or properties'}
{attribute 'enable_dynamic_creation'}
FUNCTION_BLOCK Node_F_VN_DrawRotatedRectangleExp EXTENDS VisionNode
VAR
    stRectangle : _TcVnRotatedRectangle;
    ipDestImage : _ITcVnImage;
    aColor : _TcVnVector4_LREAL;
    nThickness : _DINT(1);
    eLineType : _ETcVnLineType(ETcVnLineType.TCVN_LT_4_CONNECTED);
    hrPrev : _HRESULT(S_OK);
	hresult : _HRESULT(S_OK);
END_VAR

METHOD FB_init : BOOL
VAR_INPUT
	bInitRetains : BOOL; // if TRUE, the retain variables are initialized (warm start / cold start)
	bInCopyCode : BOOL;  // if TRUE, the instance afterwards gets moved into the copy code (online change)
END_VAR
AddInput('stRectangle', stRectangle);
AddInput('ipDestImage', ipDestImage);
AddInput('aColor', aColor);
AddParameter('nThickness', nThickness);
AddParameter('eLineType', eLineType);
AddInput('hrPrev', hrPrev);
AddOutput('ipDestImage', ipDestImage);
AddOutput('hresult',hresult);
END_METHOD

METHOD PUBLIC  Clone : I_Node
VAR
	pNode : POINTER TO Node_F_VN_DrawRotatedRectangleExp;
END_VAR
pNode := __NEW(Node_F_VN_DrawRotatedRectangleExp);
Clone := pNode^;
END_METHOD

METHOD PROTECTED OnExecute
hresult.Value := F_VN_DrawRotatedRectangleExp(
    stRectangle := stRectangle.Value,
	ipDestImage := ipDestImage.Value,
    aColor := aColor.Value,
    nThickness := nThickness.Value,
    eLineType := eLineType.Value,
	hrPrev:= hrPrev.Value);
END_METHOD

METHOD PUBLIC PreExecutionCheck
VAR_INPUT
	Check : I_PreExecutionChecks;
END_VAR
Check.IsTrue(ipDestImage.IsValid, 'ipDestImage must contain an image');
Check.IsTrue(nThickness.Value <> 0, 'nThickness must be non-zero');
END_METHOD

END_FUNCTION_BLOCK

// Nodes/Drawing/Node_F_VN_FillCircle
{attribute 'linkalways'} 
{attribute 'no_explicit_call' := 'This FB is a CLASS and must be accessed using methods or properties'}
{attribute 'enable_dynamic_creation'}
FUNCTION_BLOCK Node_F_VN_FillCircle EXTENDS VisionNode
VAR
    nCenterX : _UDINT(0);
    nCenterY : _UDINT(0);
    nRadius : _UDINT(0);
    ipDestImage : _ITcVnImage;
    aColor : _TcVnVector4_LREAL;
    hrPrev : _HRESULT(S_OK);
	hresult : _HRESULT(S_OK);
END_VAR

METHOD FB_init : BOOL
VAR_INPUT
	bInitRetains : BOOL; // if TRUE, the retain variables are initialized (warm start / cold start)
	bInCopyCode : BOOL;  // if TRUE, the instance afterwards gets moved into the copy code (online change)
END_VAR
AddParameter('nCenterX', nCenterX);
AddParameter('nCenterY', nCenterY);
AddParameter('nRadius', nRadius);
AddInput('ipDestImage', ipDestImage);
AddInput('aColor', aColor);
AddInput('hrPrev', hrPrev);
AddOutput('ipDestImage', ipDestImage);
AddOutput('hresult',hresult);
END_METHOD

METHOD PUBLIC  Clone : I_Node
VAR
	pNode : POINTER TO Node_F_VN_FillCircle;
END_VAR
pNode := __NEW(Node_F_VN_FillCircle);
Clone := pNode^;
END_METHOD

METHOD PROTECTED OnExecute
hresult.Value := F_VN_FillCircle(
    nCenterX := nCenterX.Value,
    nCenterY := nCenterY.Value,
    nRadius := nRadius.Value,
	ipDestImage := ipDestImage.Value,
    aColor := aColor.Value,
	hrPrev:= hrPrev.Value);
END_METHOD

METHOD PUBLIC PreExecutionCheck
VAR_INPUT
	Check : I_PreExecutionChecks;
END_VAR
Check.IsTrue(ipDestImage.IsValid, 'ipDestImage must contain an image');
END_METHOD

END_FUNCTION_BLOCK

// Nodes/Drawing/Node_F_VN_FillContours
{attribute 'linkalways'} 
{attribute 'no_explicit_call' := 'This FB is a CLASS and must be accessed using methods or properties'}
{attribute 'enable_dynamic_creation'}
FUNCTION_BLOCK Node_F_VN_FillContours EXTENDS VisionNode
VAR
    ipContours : _ITcVnContainer;
    nContourIndex : _DINT(0);
    ipDestImage : _ITcVnImage;
    aColor : _TcVnVector4_LREAL;
    hrPrev : _HRESULT(S_OK);
	hresult : _HRESULT(S_OK);
END_VAR

METHOD FB_init : BOOL
VAR_INPUT
	bInitRetains : BOOL; // if TRUE, the retain variables are initialized (warm start / cold start)
	bInCopyCode : BOOL;  // if TRUE, the instance afterwards gets moved into the copy code (online change)
END_VAR
AddInput('ipContours', ipContours);
AddInput('nContourIndex', nContourIndex);
AddInput('ipDestImage', ipDestImage);
AddInput('aColor', aColor);
AddInput('hrPrev', hrPrev);
AddOutput('ipDestImage', ipDestImage);
AddOutput('hresult',hresult);
END_METHOD

METHOD PUBLIC  Clone : I_Node
VAR
	pNode : POINTER TO Node_F_VN_FillContours
;
END_VAR
pNode := __NEW(Node_F_VN_FillContours);
Clone := pNode^;
END_METHOD

METHOD PROTECTED OnExecute
hresult.Value := F_VN_FillContours(
    ipContours := ipContours.Value,
    nContourIndex := nContourIndex.Value,
	ipDestImage := ipDestImage.Value,
    aColor := aColor.Value,
	hrPrev:= hrPrev.Value);
END_METHOD

METHOD PUBLIC PreExecutionCheck
VAR_INPUT
	Check : I_PreExecutionChecks;
END_VAR
VAR
    containerElements : ULINT;
    maxIndexNumber : ULINT;
END_VAR
Check.IsTrue(ipContours.IsValid, 'ipContours must be a valid container');
Check.IsTrue((ipContours.IsType(TC_GLOBAL_CONST_LIST.ContainerType_Vector_TcVnPoint2_DINT) OR
              ipContours.IsType(TC_GLOBAL_CONST_LIST.ContainerType_Vector_Vector_TcVnPoint2_DINT)),
              'ipContours contains incorrect type');

Check.IsTrue(ipContours.TryGetElementNum(containerElements) AND (containerElements > 0), 'ipContours is empty');

IF Check.Failed THEN
    RETURN;
END_IF

maxIndexNumber := containerElements - 1;

IF (nContourIndex.Value > -1) THEN
    Check.IsTrue((DINT_TO_ULINT(nContourIndex.Value) <= maxIndexNumber), 'nContourIndex out of range.');
END_IF

Check.IsTrue(ipDestImage.IsValid, 'ipDestImage must contain an image');
END_METHOD

END_FUNCTION_BLOCK

// Nodes/Drawing/Node_F_VN_FillEllipse
{attribute 'linkalways'} 
{attribute 'no_explicit_call' := 'This FB is a CLASS and must be accessed using methods or properties'}
{attribute 'enable_dynamic_creation'}
FUNCTION_BLOCK Node_F_VN_FillEllipse EXTENDS VisionNode
VAR
    stEllipse : _TcVnRotatedRectangle;
    ipDestImage : _ITcVnImage;
    aColor : _TcVnVector4_LREAL;
    hrPrev : _HRESULT(S_OK);
	hresult : _HRESULT(S_OK);
END_VAR

METHOD FB_init : BOOL
VAR_INPUT
	bInitRetains : BOOL; // if TRUE, the retain variables are initialized (warm start / cold start)
	bInCopyCode : BOOL;  // if TRUE, the instance afterwards gets moved into the copy code (online change)
END_VAR
AddInput('stEllipse', stEllipse);
AddInput('ipDestImage', ipDestImage);
AddInput('aColor', aColor);
AddInput('hrPrev', hrPrev);
AddOutput('ipDestImage', ipDestImage);
AddOutput('hresult',hresult);
END_METHOD

METHOD PUBLIC  Clone : I_Node
VAR
	pNode : POINTER TO Node_F_VN_FillEllipse;
END_VAR
pNode := __NEW(Node_F_VN_FillEllipse);
Clone := pNode^;
END_METHOD

METHOD PROTECTED OnExecute
hresult.Value := F_VN_FillEllipse(
    stEllipse := stEllipse.Value,
	ipDestImage := ipDestImage.Value,
    aColor := aColor.Value,
	hrPrev:= hrPrev.Value);
END_METHOD

METHOD PUBLIC PreExecutionCheck
VAR_INPUT
	Check : I_PreExecutionChecks;
END_VAR
Check.IsTrue(ipDestImage.IsValid, 'ipDestImage must contain an image');
END_METHOD

END_FUNCTION_BLOCK

// Nodes/Drawing/Node_F_VN_FillPolygon
{attribute 'linkalways'} 
{attribute 'no_explicit_call' := 'This FB is a CLASS and must be accessed using methods or properties'}
{attribute 'enable_dynamic_creation'}
FUNCTION_BLOCK Node_F_VN_FillPolygon EXTENDS VisionNode
VAR
    ipPoints : _ITcVnContainer;
    ipDestImage : _ITcVnImage;
    aColor : _TcVnVector4_LREAL;
    hrPrev : _HRESULT(S_OK);
	hresult : _HRESULT(S_OK);
END_VAR

METHOD FB_init : BOOL
VAR_INPUT
	bInitRetains : BOOL; // if TRUE, the retain variables are initialized (warm start / cold start)
	bInCopyCode : BOOL;  // if TRUE, the instance afterwards gets moved into the copy code (online change)
END_VAR
AddInput('ipPoints', ipPoints);
AddInput('ipDestImage', ipDestImage);
AddInput('aColor', aColor);
AddInput('hrPrev', hrPrev);
AddOutput('ipDestImage', ipDestImage);
AddOutput('hresult',hresult);
END_METHOD

METHOD PUBLIC  Clone : I_Node
VAR
	pNode : POINTER TO Node_F_VN_FillPolygon
;
END_VAR
pNode := __NEW(Node_F_VN_FillPolygon);
Clone := pNode^;
END_METHOD

METHOD PROTECTED OnExecute
hresult.Value := F_VN_FillPolygon(
    ipPoints := ipPoints.Value,
	ipDestImage := ipDestImage.Value,
    aColor := aColor.Value,
	hrPrev:= hrPrev.Value);
END_METHOD

METHOD PUBLIC PreExecutionCheck
VAR_INPUT
	Check : I_PreExecutionChecks;
END_VAR
Check.IsTrue(ipPoints.IsValid, 'ipContours must be a valid container');
Check.IsTrue((ipPoints.IsType(TC_GLOBAL_CONST_LIST.ContainerType_Vector_TcVnPoint2_DINT) OR
              ipPoints.IsType(TC_GLOBAL_CONST_LIST.ContainerType_Vector_TcVnPoint2_REAL) OR
              ipPoints.IsType(TC_GLOBAL_CONST_LIST.ContainerType_Vector_TcVnPoint2_LREAL)),
              'ipPoints contains incorrect type');

Check.IsTrue(ipDestImage.IsValid, 'ipDestImage must contain an image');
END_METHOD

END_FUNCTION_BLOCK

// Nodes/Drawing/Node_F_VN_FillRectangle
{attribute 'linkalways'} 
{attribute 'no_explicit_call' := 'This FB is a CLASS and must be accessed using methods or properties'}
{attribute 'enable_dynamic_creation'}
FUNCTION_BLOCK Node_F_VN_FillRectangle EXTENDS VisionNode
VAR
    nTopLeftX : _UDINT(0);
    nTopLeftY : _UDINT(0);
    nBottomRightX : _UDINT(0);
    nBottomRightY : _UDINT(0);
    ipDestImage : _ITcVnImage;
    aColor : _TcVnVector4_LREAL;
    hrPrev : _HRESULT(S_OK);
	hresult : _HRESULT(S_OK);
END_VAR

METHOD FB_init : BOOL
VAR_INPUT
	bInitRetains : BOOL; // if TRUE, the retain variables are initialized (warm start / cold start)
	bInCopyCode : BOOL;  // if TRUE, the instance afterwards gets moved into the copy code (online change)
END_VAR
AddParameter('nTopLeftX', nTopLeftX);
AddParameter('nTopLeftY', nTopLeftY);
AddParameter('nBottomRightX', nBottomRightX);
AddParameter('nBottomRightY', nBottomRightY);
AddInput('ipDestImage', ipDestImage);
AddInput('aColor', aColor);
AddInput('hrPrev', hrPrev);
AddOutput('ipDestImage', ipDestImage);
AddOutput('hresult',hresult);
END_METHOD

METHOD PUBLIC  Clone : I_Node
VAR
	pNode : POINTER TO Node_F_VN_FillRectangle;
END_VAR
pNode := __NEW(Node_F_VN_FillRectangle);
Clone := pNode^;
END_METHOD

METHOD PROTECTED OnExecute
hresult.Value := F_VN_FillRectangle(
    nTopLeftX := nTopLeftX.Value,
    nTopLeftY := nTopLeftY.Value,
    nBottomRightX := nBottomRightX.Value,
    nBottomRightY := nBottomRightY.Value,
	ipDestImage := ipDestImage.Value,
    aColor := aColor.Value,
	hrPrev:= hrPrev.Value);
END_METHOD

METHOD PUBLIC PreExecutionCheck
VAR_INPUT
	Check : I_PreExecutionChecks;
END_VAR
Check.IsTrue(ipDestImage.IsValid, 'ipDestImage must contain an image');
END_METHOD

END_FUNCTION_BLOCK

// Nodes/Drawing/Node_F_VN_FillRotatedRectangle
{attribute 'linkalways'} 
{attribute 'no_explicit_call' := 'This FB is a CLASS and must be accessed using methods or properties'}
{attribute 'enable_dynamic_creation'}
FUNCTION_BLOCK Node_F_VN_FillRotatedRectangle EXTENDS VisionNode
VAR
    stRectangle : _TcVnRotatedRectangle;
    ipDestImage : _ITcVnImage;
    aColor : _TcVnVector4_LREAL;
    hrPrev : _HRESULT(S_OK);
	hresult : _HRESULT(S_OK);
END_VAR

METHOD FB_init : BOOL
VAR_INPUT
	bInitRetains : BOOL; // if TRUE, the retain variables are initialized (warm start / cold start)
	bInCopyCode : BOOL;  // if TRUE, the instance afterwards gets moved into the copy code (online change)
END_VAR
AddInput('stRectangle', stRectangle);
AddInput('ipDestImage', ipDestImage);
AddInput('aColor', aColor);
AddInput('hrPrev', hrPrev);
AddOutput('ipDestImage', ipDestImage);
AddOutput('hresult',hresult);
END_METHOD

METHOD PUBLIC  Clone : I_Node
VAR
	pNode : POINTER TO Node_F_VN_FillRotatedRectangle;
END_VAR
pNode := __NEW(Node_F_VN_FillRotatedRectangle);
Clone := pNode^;
END_METHOD

METHOD PROTECTED OnExecute
hresult.Value := F_VN_FillRotatedRectangle(
    stRectangle := stRectangle.Value,
	ipDestImage := ipDestImage.Value,
    aColor := aColor.Value,
	hrPrev:= hrPrev.Value);
END_METHOD

METHOD PUBLIC PreExecutionCheck
VAR_INPUT
	Check : I_PreExecutionChecks;
END_VAR
Check.IsTrue(ipDestImage.IsValid, 'ipDestImage must contain an image');
END_METHOD

END_FUNCTION_BLOCK

// Nodes/Drawing/Node_F_VN_PlotIntensityProfile
{attribute 'linkalways'} 
{attribute 'no_explicit_call' := 'This FB is a CLASS and must be accessed using methods or properties'}
{attribute 'enable_dynamic_creation'}
FUNCTION_BLOCK Node_F_VN_PlotIntensityProfile EXTENDS VisionNode
VAR
    ipSrcImage : _ITcVnImage;
    ipDestImage : _ITcVnImage;
    aStartPoint : _TcVnPoint2_REAL;
    aEndPoint : _TcVnPoint2_REAL;
    hrPrev : _HRESULT(S_OK);
	hresult : _HRESULT(S_OK);
END_VAR

METHOD FB_init : BOOL
VAR_INPUT
	bInitRetains : BOOL; // if TRUE, the retain variables are initialized (warm start / cold start)
	bInCopyCode : BOOL;  // if TRUE, the instance afterwards gets moved into the copy code (online change)
END_VAR
AddInput('ipSrcImage', ipSrcImage);
AddInput('aStartPoint', aStartPoint);
AddInput('aEndPoint', aEndPoint);
AddInput('hrPrev', hrPrev);
AddOutput('ipDestImage', ipDestImage);
AddOutput('hresult',hresult);
END_METHOD

METHOD PUBLIC  Clone : I_Node
VAR
	pNode : POINTER TO Node_F_VN_PlotIntensityProfile;
END_VAR
pNode := __NEW(Node_F_VN_PlotIntensityProfile);
Clone := pNode^;
END_METHOD

METHOD PROTECTED OnExecute
hresult.Value := F_VN_PlotIntensityProfile(
	ipSrcImage := ipSrcImage.Value,
    ipDestImage := ipDestImage.Value,
    aStartPoint := aStartPoint.Value,
    aEndPoint := aEndPoint.Value,
	hrPrev:= hrPrev.Value);
END_METHOD

METHOD PUBLIC PreExecutionCheck
VAR_INPUT
	Check : I_PreExecutionChecks;
END_VAR
Check.IsTrue(ipSrcImage.IsValid, 'ipSrcImage must contain an image');
Check.IsTrue(ipSrcImage.HasChannelCount(1), 'ipSrcImage must have 1 channel');
Check.IsTrue(ipSrcImage.IsPixelDepth(8), 'ipSrcImage must have 8 bit pixel depth');
END_METHOD

END_FUNCTION_BLOCK

